(* Trigger ********************************************************)

(* Bausteine ******************************************************)
	Event													:	EventHandlingGrp10 := (
																	AutoConfirm			:= FALSE, 
																	SetClass 			:= TC2_SYSTEM.TCEVENTCLASS_ALARM );
	ChnEvent												:	NciChnEventHandling;

(* Dummy Speicher *************************************************)
	i														:	INT ;

END_VAR

(* Error message NCI channel to EventLogger 	V1.0	DS	*)
(***********************************************************)

(* Sequence **************************************************************)
IF __ISVALIDREF(rNci) 
THEN
	(* get Quit signal **************************************************)
	IF ConfirmTrig 
	THEN 
		QuitInternal 										:= TRUE; 
	END_IF (* set false see below *)

(* Event Logger Meldungen *****************************************************)
	Event.no[1].Flag 										:= rNci.IsEStopRequested;
	Event.no[2].Flag 										:= rNci.IsFeedFromBackupList;   
	Event.no[3].Flag 										:= rNci.IsMovingBackward;   
	
(*
	Event.no[4].Flag 										:= FALSE;
	Event.no[5].Flag 										:= FALSE;
	Event.no[6].Flag 										:= FALSE;
	Event.no[7].Flag 										:= FALSE;
	Event.no[8].Flag 										:= FALSE;
	Event.no[9].Flag 										:= FALSE;
	Event.no[10].Flag 										:= FALSE;
*)
(* workl Event Ctrl *************************************************)
	IF Event.no[1].Text2 <> Name OR Event.no[1].Text2 <> ''
	THEN
		//Init EventClass
		Event.no[1].eClass 									:= TC2_SYSTEM.TCEVENTCLASS_HINT;
		Event.no[2].eClass 									:= TC2_SYSTEM.TCEVENTCLASS_STATEINFO;
		Event.no[3].eClass 									:= TC2_SYSTEM.TCEVENTCLASS_STATEINFO;

		(* Init Name *)
		FOR i := Event.MIN_EVENT TO Event.MAX_EVENT DO
			Event.no[i].Text2								:= SEL(LEN(name)>1,CONCAT('Channel id:',DWORD_TO_STRING(rNci.NciToPlc.ChnId)),name);
		END_FOR
	END_IF

	Event(
		ConfirmTrig := ConfirmTrig,
		Disable		:= NOT Enable,
		SourceId	:= SourceId + rNci.NciToPlc.ChnId,
		Status	 	=> );	

(* Send ErrorId Message Text **********************************)
	ChnEvent(
		ConfirmTrig	:= NOT Enable OR QuitInternal OR ErrorId = 0 AND ChnEvent.State <> 0,
		Name		:= name,
		ChannelId	:= rNci.NciToPlc.ChnId,
		SourceId	:= Event.SourceId,
		Flag		:= ErrorId > 0 AND Enable,
		ErrorID		:= ErrorId,
		State		=> );

(* EventStatus *************************************************)
	Status													:= ChnEvent.Status OR Event.Status;
	NoOfActiveEvents										:= Event.NoOfActiveEvents + SEL(ChnEvent.Status.31 , 0, 1);

(* Error unkonw pointer or channel id *****************************)
ELSE
	NoOfActiveEvents										:= 0;
	ChnEvent(Flag := FALSE, ConfirmTrig := ChnEvent.State <> 0);
	Event(Disable := TRUE, Status =>  ); 
	Status													:= ChnEvent.Status OR Event.Status;
END_IF

(* Default reset Quit Internal *******************************)
	QuitInternal 											:= FALSE;

(**************************************************************)

METHOD PUBLIC confirm : bool  //Return value = TRUE if execution finished 
VAR_INPUT
END_VAR
QuitInternal 												:= TRUE;
confirm														:= TRUE;
END_METHOD

END_FUNCTION_BLOCK

// POUs/Motion/TF5100-NCI/02_Options/MFunctions/NciMFnc
{attribute 'no_check'}
FUNCTION_BLOCK NciMFnc
VAR_OUTPUT CONSTANT 
	MIN_M_FUNC												:	 UINT := 0;
	MAX_M_FUNC												:	 UINT := 159;
	
//Predefined M Functions
	M2_PRG_END												:	UINT := 2;
	M17_END_SUBROUTINE										:	UINT := 17;
	M30_PRG_END_WITH_ALL_MFUNC								:	UINT := 30; 
END_VAR                 									
VAR_INPUT               									
	ConfirmHsk												:	BOOL := FALSE; (* oder Methode benutzen *)
	FastMFuncReset											:	BOOL := FALSE; (* Signal Start Reser der unter FastMFuncNo angegebenen MFunc Nr. *)
	FastMFuncNo												:	UINT (MIN_M_FUNC..MAX_M_FUNC) := MIN_M_FUNC; (* Nr. der MFunktion die Resetet werden soll *)
	rNCIRef													:	REFERENCE TO NCI_REF := 0;
END_VAR                 									
VAR_OUTPUT              	
	HskReq													:	BOOL;
	HskId													:	UINT; 	
	CntActive												:	INT; //Count number of active M fucntions
	Active													:	BOOL; //Rising trigger M-Function active
	No														:	ARRAY[MIN_M_FUNC..MAX_M_FUNC] OF BOOL; (* Array of M-Functions *)
	rtNo													:	ARRAY[MIN_M_FUNC..MAX_M_FUNC] OF BOOL; (* rising trigger of M-Functions *)
END_VAR                     								
VAR
(* Zwischenspeicher ************************************************************)
	MemFnc													:	INT := -1;

(* Deklaration Trigger **********************************************************)

(* Zeiten ******************************************************************)

(* Bausteine ***************************************************************)
	ItpResetFastMFuncEx										:  ItpResetFastMFuncEx := (tTimeOut	:= DEFAULT_ADS_TIMEOUT);

(* Dummy Speicher **********************************************************)
	i														:	UINT := 0;
	OK														:	BOOL;
END_VAR

	(************************************************************************************)
	(*																					*)
	(*		B E C K H O F F   N E W   A U T O M A T I O N   T E C H N O L O G Y    		*)
	(*																					*)
	(*		Eiserstr.5	D-33415 Verl	Germany	phone:	+49-5246-0	www.Beckhoff.Com	*)
    (*																					*)
    (*		Bausteinbeschreibung	:	Auswerten von M-Funktionen						*)
	(*		TwinCAT-Version			:	2.11.x 											*)
	(*		Version					:	V2.0/ 05/20										*)
 	(*		Autor					:	Daniel Schlingmann								*)
	(*		Lib						:	TcNCI.Lib										*)
	(*																					*)
	(************************************************************************************)

(* evaluate M-function with additional acknowledge *********************************************************************)
	HskReq 													:= rNCIRef.NciToPlc.HskMFuncReq.0;
	HskId 													:= SEL(HskReq, 0, rNCIRef.NciToPlc.HskMFuncNo);

	(* Confirm request *)
	rNCIRef.PlcToNci.MFuncGranted.0 						:= (ConfirmHsk OR rNCIRef.PlcToNci.MFuncGranted.0) AND rNCIRef.NciToPlc.HskMFuncReq.0;

(* set all M-function setzen *)
	CntActive												:= 0;
	Active													:= FALSE;
	
	FOR i := MIN_M_FUNC TO MAX_M_FUNC DO
	 	OK	 												:= ItpIsFastMFunc(UINT_TO_INT(i),rNCIRef.NciToPlc) OR rNCIRef.NciToPlc.HskMFuncNo = i AND rNCIRef.NciToPlc.HskMFuncReq.0;
		rtNo[i]												:= NOT No[i] AND OK;
		No[i]												:= OK;
		IF No[i] 
		THEN 
			CntActive										:= CntActive + 1;		
			Active 											:= TRUE; 
		END_IF
	END_FOR

(* reset fast M-functions, ResetFastMFunc can also be used *)
	IF MemFnc < 0
	THEN
		IF FastMFuncReset
		THEN
			MemFnc 											:= 1;
			ResetFastMFunc(FastMFuncNo:= FastMFuncNo);
		END_IF
	ELSE 
		ResetFastMFunc(FastMFuncNo:= FastMFuncNo);		
	END_IF

(************************************************************************************)

METHOD PUBLIC confirm : BOOL //Return value = TRUE if execution finished
//required parameter
//rNCIRef
VAR_INPUT
END_VAR
IF __ISVALIDREF(rNCIRef)
THEN
	rNCIRef.PlcToNci.MFuncGranted.0 						:= rNCIRef.NciToPlc.HskMFuncReq.0;
	Confirm													:= NOT rNCIRef.NciToPlc.HskMFuncReq.0;
ELSE
	Confirm 												:= TRUE;
END_IF
END_METHOD

METHOD PUBLIC resetFastMFunc : BOOL //Return value = TRUE if busy
//required parameter
//rNCIRef
VAR_INPUT
	FastMFuncNo												:	UINT; (* number of M-function, which has to be resetted *)
END_VAR
IF NOT __ISVALIDREF(rNCIRef)
THEN
	ResetFastMFunc											:= FALSE;
	Return;	
END_IF

	IF ItpIsFastMFunc(UINT_TO_INT(FastMFuncNo),rNCIRef.NciToPlc) 
	THEN
		ItpResetFastMFuncEx.bExecute 						:= TRUE;
		MemFnc.0											:= TRUE;
	ELSIF NOT ItpResetFastMFuncEx.bBusy             		
	THEN                                            		
		ItpResetFastMFuncEx.bExecute 						:= FALSE;
	END_IF
	
	THIS^.FastMFuncNo										:= FastMFuncNo;

	ItpResetFastMFuncEx(
		bExecute	:= ,
		nMFuncNo	:= FastMFuncNo,
		tTimeOut	:= ,
		sNciToPlc	:= rNCIRef.NciToPlc,
		bBusy		=> ,
		bErr		=> ,
		nErrId	=> );
		
	IF NOT ItpResetFastMFuncEx.bBusy
	THEN
		IF ItpResetFastMFuncEx.bExecute
		THEN
			;
		//	Error											:=	ItpResetFastMFuncEx.bErr;
		//	ErrorId											:= ItpResetFastMFuncEx.nErrId;
		END_IF
		IF NOT ItpIsFastMFunc(UINT_TO_INT(FastMFuncNo),rNCIRef.NciToPlc) 
		THEN
			MemFnc											:= -1;
			ItpResetFastMFuncEx(bExecute := FALSE , sNciToPlc:= rNCIRef.NciToPlc);
		END_IF
	END_IF
	
	resetFastMFunc											:= ItpResetFastMFuncEx.bBusy;
END_METHOD

END_FUNCTION_BLOCK

// POUs/Motion/TF5100-NCI/02_Options/PlcItp/NciCreateItpTable
{attribute 'no_check'}
//Create Nci PlcInterpolation tabel
//
FUNCTION_BLOCK NciCreateItpTable
VAR_INPUT
	BlockNo													: UDINT := 0; //Block number addtional parameter for methods. At 0 -> block number will be automatically increased by every new entry
	OffsetFactorTblNumber									: UDINT := 100; 
	MaxTblNumber											: UDINT := 1000; 
END_VAR                     								
VAR_OUTPUT                  								
	Table													: ST_NciFeedGroupTable;
	FilledRows												: INT;
	LastBlockNo												: UDINT; //Last Blocknumber 
	Error													: BOOL;
{attribute 'displaymode':='hex'}
	ErrorID													: UDINT;
	ErrorText												: STRING(20);
END_VAR                     								
VAR
// Cache *******************************************
	TableNumber												: UDINT := 0;
	BlockCount												: UDINT := 1;

// Timer ******************************************************
// Trigger ****************************************************
// Blocks *****************************************************
	TblTemplate												: NciCreateItpTableEntryTemplate;
// Error ******************************************************
// Dummy Speicher *********************************************
	i														: INT := 0;
END_VAR

(* writing TcPlcInterpolation table				V1.5	*)
(********************************************************)

(* pleas use methods instead of the function-block body ********************)
	;
(***************************************************************************)

METHOD addCircleCIP : BOOL //Return value = TRUE if executed succesful
VAR_INPUT
	X														: LREAL := 0.0;
	Y														: LREAL := 0.0;
	Z														: LREAL := 0.0;
	Q1														: LREAL := 0.0;
	Q2														: LREAL := 0.0;
	Q3														: LREAL := 0.0;
	Q4														: LREAL := 0.0;
	Q5														: LREAL := 0.0;
	Velo													: LREAL; 	// mm/s 
	AccurateStop											: BOOL := FALSE;
	CIPPosX													: LREAL := 0.0;
	CIPPosY													: LREAL := 0.0;
	CIPPosZ													: LREAL := 0.0;
END_VAR
	(* NCI GeoCirclePlane schreiben									*)
	(*********************************************************)

(* Zielpos. in Tabelle schreiben ************************************************************)
	BlockCount 												:= BlockCount + 1;
	TblTemplate.GeoCircleCIP.nDisplayIndex := LastBlockNo 	:= SEL(BlockNo = 0, BlockNo, TableNumber * OffsetFactorTblNumber + BlockCount);
	TblTemplate.GeoCircleCIP.fEndPosX						:= X;
	TblTemplate.GeoCircleCIP.fEndPosY						:= Y;
	TblTemplate.GeoCircleCIP.fEndPosZ						:= Z;
	TblTemplate.GeoCircleCIP.fEndPosQ1						:= Q1;
	TblTemplate.GeoCircleCIP.fEndPosQ2						:= Q2;
	TblTemplate.GeoCircleCIP.fEndPosQ3						:= Q3;
	TblTemplate.GeoCircleCIP.fEndPosQ4						:= Q4;
	TblTemplate.GeoCircleCIP.fEndPosQ5						:= Q5;
	TblTemplate.GeoCircleCIP.fVelo							:= Velo;
	TblTemplate.GeoCircleCIP.bAccurateStop					:= AccurateStop;
	TblTemplate.GeoCircleCIP.fCIPPosX						:= CIPPosX;
	TblTemplate.GeoCircleCIP.fCIPPosY						:= CIPPosY;
	TblTemplate.GeoCircleCIP.fCIPPosZ						:= CIPPosZ;
                                                        	
	TblTemplate.InsertGeoCircleCIP(Table:= Table);    	
	Error													:= TblTemplate.Error;
	ErrorId													:= TblTemplate.ErrorId;
	ErrorText												:= TblTemplate.ErrorText;
	FilledRows												:= TblTemplate.FilledRows;

	AddCircleCip											:= NOT Error;
(***************************************************************************)
END_METHOD

METHOD addDwellTime : BOOL //Return value = TRUE if executed succesful
VAR_INPUT
	/// UCS ObjectID 
	Value													: LREAL ;
END_VAR
(*  													*)
(********************************************************)
	BlockCount 												:= BlockCount + 1;
	TblTemplate.DwellTime.nDisplayIndex	 := LastBlockNo 	:= SEL(BlockNo = 0, BlockNo, TableNumber * OffsetFactorTblNumber + BlockCount);
	TblTemplate.DwellTime.fDwellTime						:= Value;

	TblTemplate.InsertDwellTime(Table:= Table);
	Error													:= TblTemplate.Error;
	ErrorId													:= TblTemplate.ErrorId;
	ErrorText												:= TblTemplate.ErrorText;
	FilledRows												:= TblTemplate.FilledRows;

	AddDwellTime											:= not Error;	
	

(***************************************************************************)
END_METHOD

METHOD addEndOfTable : BOOL //Return value = TRUE if executed succesful
TblTemplate.InsertEndOfTable(Table:= Table);
Error													:= TblTemplate.Error;
ErrorId													:= TblTemplate.ErrorId;
ErrorText												:= TblTemplate.ErrorText;
FilledRows												:= TblTemplate.FilledRows;

AddEndOfTable											:= NOT Error;
END_METHOD

METHOD addMFuncFast : BOOL //Return value = TRUE if executed succesful
VAR_INPUT
	MFuncNo													: INT := 0;
END_VAR
(*														*)
(********************************************************)

(*************************************************************************************)
	BlockCount 												:= BlockCount + 1;
	TblTemplate.MFuncFast.nDisplayIndex := LastBlockNo 		:= SEL(BlockNo = 0, BlockNo, TableNumber * OffsetFactorTblNumber + BlockCount);
	TblTemplate.MFuncFast.nMFuncIn0							:= MFuncNo;
	TblTemplate.MFuncFast.nMFuncIn1							:= -1;
	TblTemplate.MFuncFast.nMFuncIn2							:= -1;
	TblTemplate.MFuncFast.nMFuncIn3							:= -1;
	TblTemplate.MFuncFast.nMFuncIn4							:= -1;
	TblTemplate.MFuncFast.nMFuncIn5							:= -1;
	TblTemplate.MFuncFast.nMFuncIn6							:= -1;
	TblTemplate.MFuncFast.nMFuncIn7							:= -1;
	
	TblTemplate.InsertMFuncFast(Table:= Table);
	Error													:= TblTemplate.Error;
	ErrorId													:= TblTemplate.ErrorId;
	ErrorText												:= TblTemplate.ErrorText;
	FilledRows												:= TblTemplate.FilledRows;
	
	AddMFuncFast											:= not Error;
(*************************************************************************************)
END_METHOD

METHOD addMFuncFastList : BOOL //Return value = TRUE if executed succesful
VAR_INPUT
	MFuncNo0												: INT := -1; //0-159 > Set to -1 to mark end of used MFunc
	MFuncNo1												: INT := -1; //0-159 > Set to -1 to mark end of used MFunc
	MFuncNo2												: INT := -1; //0-159 > Set to -1 to mark end of used MFunc
	MFuncNo3												: INT := -1; //0-159 > Set to -1 to mark end of used MFunc
	MFuncNo4												: INT := -1; //0-159 > Set to -1 to mark end of used MFunc
	MFuncNo5												: INT := -1; //0-159 > Set to -1 to mark end of used MFunc
	MFuncNo6												: INT := -1; //0-159 > Set to -1 to mark end of used MFunc
	MFuncNo7												: INT := -1; //0-159 > Set to -1 to mark end of used MFunc
END_VAR
(*														*)
(********************************************************)

(*************************************************************************************)
	BlockCount 												:= BlockCount + 1;
	TblTemplate.MFuncFast.nDisplayIndex := LastBlockNo 		:= SEL(BlockNo = 0, BlockNo, TableNumber * OffsetFactorTblNumber + BlockCount);
	TblTemplate.MFuncFast.nMFuncIn0							:= MFuncNo0;
	TblTemplate.MFuncFast.nMFuncIn1							:= MFuncNo1;
	TblTemplate.MFuncFast.nMFuncIn2							:= MFuncNo2;
	TblTemplate.MFuncFast.nMFuncIn3							:= MFuncNo3;
	TblTemplate.MFuncFast.nMFuncIn4							:= MFuncNo4;
	TblTemplate.MFuncFast.nMFuncIn5							:= MFuncNo5;
	TblTemplate.MFuncFast.nMFuncIn6							:= MFuncNo6;
	TblTemplate.MFuncFast.nMFuncIn7							:= MFuncNo7;
	
	TblTemplate.InsertMFuncFast(Table:= Table);
	Error													:= TblTemplate.Error;
	ErrorId													:= TblTemplate.ErrorId;
	ErrorText												:= TblTemplate.ErrorText;
	FilledRows												:= TblTemplate.FilledRows;
	
	AddMFuncFastList										:= NOT Error;
(*************************************************************************************)
END_METHOD

METHOD addMFuncHsk : BOOL //Return value = TRUE if executed succesful
VAR_INPUT
	MFuncNo													: INT := 0;
END_VAR
(* 														*)
(********************************************************)

(*************************************************************************************)
	BlockCount 												:= BlockCount + 1;
	TblTemplate.MFuncHsk.nDisplayIndex := LastBlockNo 		:= SEL(BlockNo = 0, BlockNo,  TableNumber * OffsetFactorTblNumber + BlockCount);
	TblTemplate.MFuncHsk.nMFunc								:= MFuncNo;
                                                        	
	TblTemplate.InsertMFuncHsk(Table:= Table);          	
	Error													:= TblTemplate.Error;
	ErrorId													:= TblTemplate.ErrorId;
	ErrorText												:= TblTemplate.ErrorText;
	FilledRows												:= TblTemplate.FilledRows;
	
	AddMFuncHsk												:= not Error;
(*************************************************************************************)
END_METHOD

METHOD addMFuncResetAllFast : BOOL //Return value = TRUE if executed succesful
VAR_INPUT
END_VAR
(* NCI ResetAllFastMFunc schreiben								*)
(*************************************************************************************)

(* confirmError all fast M-functions****************************************************)
	BlockCount 													:= BlockCount + 1;
	TblTemplate.MFuncResetAllFast.nDisplayIndex	:= LastBlockNo 	:= SEL(BlockNo = 0, BlockNo, TableNumber * OffsetFactorTblNumber + BlockCount);
	TblTemplate.InsertMFuncResetAllFast(Table:= Table);
	Error														:= TblTemplate.Error;
	ErrorId														:= TblTemplate.ErrorId;
	ErrorText													:= TblTemplate.ErrorText;
	FilledRows													:= TblTemplate.FilledRows;
	
	AddMFuncResetAllFast										:= not Error;
(*************************************************************************************)
END_METHOD

METHOD reset : BOOL //Return value = TRUE if execution finished
VAR_INPUT
END_VAR
TblTemplate.Reset(Table := Table);
FilledRows													:= 0;
BlockCount 													:= 0;
LastBlockNo													:= 0;
TableNumber 												:= TableNumber + 1;

IF TableNumber > MaxTblNumber 
THEN 
	TableNumber 											:= 1; 
END_IF

Error 														:= FALSE;
Errorid														:= 0;
ErrorText													:= '';
Reset														:= TRUE;
END_METHOD

METHOD setAxisDynamics : bool //Return value = TRUE if executed succesful
VAR_INPUT
	AxisNo													:	UDINT;
	Acc,Dec,Jerk											:	LREAL;
END_VAR
	(* NCI SetAxisDynamics schreiben						*)
	(*********************************************************)

(* Zielpos. in Tabelle schreiben ************************************************************)
	BlockCount 												:= BlockCount + 1;
	TblTemplate.AxisDynamics.nDisplayIndex := LastBlockNo := SEL(BlockNo = 0, BlockNo, TableNumber * OffsetFactorTblNumber + BlockCount);

	TblTemplate.AxisDynamics.nAxis 							:= AxisNo;
	TblTemplate.AxisDynamics.fDec							:= Dec;
	TblTemplate.AxisDynamics.fJerk							:= Jerk;
	TblTemplate.AxisDynamics.fAcc							:= Acc;
                                                        	
	TblTemplate.InsertAxisDynamics(Table:= Table);    	
	Error													:= TblTemplate.Error;
	ErrorId													:= TblTemplate.ErrorId;
	ErrorText												:= TblTemplate.ErrorText;
	FilledRows												:= TblTemplate.FilledRows;

	SetAxisDynamics											:= NOT Error;
(***************************************************************************)
END_METHOD

METHOD setBaseFrame : bool //Return value = TRUE if executed succesful
VAR_INPUT
    ShiftX													: LREAL;
    ShiftY													: LREAL;
    ShiftZ													: LREAL;
    RotX													: LREAL;
    RotY													: LREAL;
    RotZ													: LREAL;
    ShiftQ1													: LREAL;
    ShiftQ2													: LREAL;
    ShiftQ3													: LREAL;
    ShiftQ4													: LREAL;
    ShiftQ5													: LREAL;
END_VAR
	(* NCI SetBaseFrame schreiben						*)
	(*********************************************************)

(* Zielpos. in Tabelle schreiben ************************************************************)
	BlockCount 												:= BlockCount + 1;
	TblTemplate.BaseFrame.nDisplayIndex := LastBlockNo := SEL(BlockNo = 0, BlockNo, TableNumber * OffsetFactorTblNumber + BlockCount);

    TblTemplate.BaseFrame.fShiftX 							:= ShiftX;
    TblTemplate.BaseFrame.fShiftY							:= ShiftY;
    TblTemplate.BaseFrame.fShiftZ							:= ShiftZ;
    TblTemplate.BaseFrame.fRotX								:= RotX;
    TblTemplate.BaseFrame.fRotY								:= RotY;
    TblTemplate.BaseFrame.fRotZ								:= RotZ;
    TblTemplate.BaseFrame.fShiftQ1							:= ShiftQ1;
    TblTemplate.BaseFrame.fShiftQ2							:= ShiftQ2;
    TblTemplate.BaseFrame.fShiftQ3							:= ShiftQ3;
    TblTemplate.BaseFrame.fShiftQ4							:= ShiftQ4;
    TblTemplate.BaseFrame.fShiftQ5							:= ShiftQ5;
                       	
	TblTemplate.InsertBaseFrame(Table:= Table);    	
	Error													:= TblTemplate.Error;
	ErrorId													:= TblTemplate.ErrorId;
	ErrorText												:= TblTemplate.ErrorText;
	FilledRows												:= TblTemplate.FilledRows;

	SetBaseFrame											:= NOT Error;
(***************************************************************************)
END_METHOD

METHOD setCirclePlane : BOOL //Return value = TRUE if executed succesful
VAR_INPUT
	X														: LREAL := 0.0;
	Y														: LREAL := 0.0;
	Z														: LREAL := 0.0;
	Q1														: LREAL := 0.0;
	Q2														: LREAL := 0.0;
	Q3														: LREAL := 0.0;
	Q4														: LREAL := 0.0;
	Q5														: LREAL := 0.0;
	Velo													: LREAL; 	// mm/s 
	AccurateStop											: BOOL := FALSE;
	Clockwise												: BOOL := TRUE;
	Plane													: E_NciGeoPlane := E_NciGeoPlaneXY;
	CenterX													: LREAL := 0.0;
	CenterY													: LREAL := 0.0;
	CenterZ													: LREAL := 0.0;
END_VAR
	(* NCI GeoCirclePlane schreiben									*)
	(*********************************************************)

(* Zielpos. in Tabelle schreiben ************************************************************)
	BlockCount 												:= BlockCount + 1;
	TblTemplate.GeoCirclePlane.nDisplayIndex := LastBlockNo := SEL(BlockNo = 0, BlockNo, TableNumber * OffsetFactorTblNumber + BlockCount);
	TblTemplate.GeoCirclePlane.fEndPosX						:= X;
	TblTemplate.GeoCirclePlane.fEndPosY						:= Y;
	TblTemplate.GeoCirclePlane.fEndPosZ						:= Z;
	TblTemplate.GeoCirclePlane.fEndPosQ1					:= Q1;
	TblTemplate.GeoCirclePlane.fEndPosQ2					:= Q2;
	TblTemplate.GeoCirclePlane.fEndPosQ3					:= Q3;
	TblTemplate.GeoCirclePlane.fEndPosQ4					:= Q4;
	TblTemplate.GeoCirclePlane.fEndPosQ5					:= Q5;
	TblTemplate.GeoCirclePlane.fVelo						:= Velo;
	TblTemplate.GeoCirclePlane.bAccurateStop				:= AccurateStop;
	TblTemplate.GeoCirclePlane.bClockwise					:= Clockwise;
	TblTemplate.GeoCirclePlane.nPlane						:= Plane;
	TblTemplate.GeoCirclePlane.fCenterX						:= CenterX;
	TblTemplate.GeoCirclePlane.fCenterY						:= CenterY;
	TblTemplate.GeoCirclePlane.fCenterZ						:= CenterZ;
                                                        	
	TblTemplate.InsertGeoCirclePlane(Table:= Table);    	
	Error													:= TblTemplate.Error;
	ErrorId													:= TblTemplate.ErrorId;
	ErrorText												:= TblTemplate.ErrorText;
	FilledRows												:= TblTemplate.FilledRows;

	SetCirclePlane											:= NOT Error;
(***************************************************************************)
END_METHOD

METHOD setCoordinateSystem : BOOL //Return value = TRUE if executed succesful
VAR_INPUT
	/// UCS ObjectID 
	ObjectId												: UDINT := 0;
END_VAR
(* NCI UserKos schreiben															*)
(************************************************************************************)

(* User Koordinatensystem schreiben ************************************************************)
	BlockCount 												:= BlockCount + 1;
	TblTemplate.SetCoordinateSystem.nDisplayIndex := LastBlockNo := SEL(BlockNo = 0, BlockNo, TableNumber * OffsetFactorTblNumber + BlockCount);
	TblTemplate.SetCoordinateSystem.nObjectId				:= ObjectId;

	TblTemplate.InsertSetCoordinateSystem(Table:= Table);
	Error													:= TblTemplate.Error;
	ErrorId													:= TblTemplate.ErrorId;
	ErrorText												:= TblTemplate.ErrorText;
	FilledRows												:= TblTemplate.FilledRows;
	
	SetCoordinateSystem										:= not Error;
(*************************************************************************************)
END_METHOD

METHOD setDynOverride : BOOL //Return value = TRUE if executed succesful
VAR_INPUT
	/// UCS ObjectID 
	Value													: lreal := 0; //0.0-100.0%
END_VAR
(* NCI Oevrride schreiben											*)
(********************************************************************)

(* insert override **************************************************)
	(* apapt override *)
	BlockCount 												:= BlockCount + 1;
	TblTemplate.DynOverride.nDisplayIndex := LastBlockNo 		:= SEL(BlockNo = 0, BlockNo, TableNumber * OffsetFactorTblNumber + BlockCount);
	TblTemplate.DynOverride.fDynOvr								:= 0.01 * Value;

	TblTemplate.InsertDynOverride(Table:= Table);
	Error													:= TblTemplate.Error;
	ErrorId													:= TblTemplate.ErrorId;
	ErrorText												:= TblTemplate.ErrorText;
	FilledRows												:= TblTemplate.FilledRows;
	
	SetDynOverride											:= not Error;
(*************************************************************************************)
END_METHOD

METHOD setGeoBezier3 : booL //Return value = TRUE if executed succesful
VAR_INPUT
     ControlPoint1X											: LREAL;
     ControlPoint1Y											: LREAL;
     ControlPoint1Z											: LREAL;
     ControlPoint2X											: LREAL;
     ControlPoint2Y											: LREAL;
     ControlPoint2Z											: LREAL;
     EndPosX												: LREAL;
     EndPosY												: LREAL;
     EndPosZ												: LREAL;
     EndPosQ1												: LREAL;
     EndPosQ2												: LREAL;
     EndPosQ3												: LREAL;
     EndPosQ4												: LREAL;
     EndPosQ5												: LREAL;
     Velo													: LREAL;
     AccurateStop											: BOOL; (* VeloEnd := 0 *)
END_VAR
	(* NCI SetGeoBezier3 schreiben						*)
	(*********************************************************)

(* Zielpos. in Tabelle schreiben ************************************************************)
	BlockCount 												:= BlockCount + 1;
	TblTemplate.GeoBezier3.nDisplayIndex := LastBlockNo := SEL(BlockNo = 0, BlockNo, TableNumber * OffsetFactorTblNumber + BlockCount);

    TblTemplate.GeoBezier3.fControlPoint1X					:= ControlPoint1X;
    TblTemplate.GeoBezier3.fControlPoint1Y					:= ControlPoint1Y;
    TblTemplate.GeoBezier3.fControlPoint1Z					:= ControlPoint1Z;
    TblTemplate.GeoBezier3.fControlPoint2X					:= ControlPoint2X;
    TblTemplate.GeoBezier3.fControlPoint2Y					:= ControlPoint2Y;
    TblTemplate.GeoBezier3.fControlPoint2Z					:= ControlPoint2Z;
    TblTemplate.GeoBezier3.fEndPosX							:= EndPosX;
    TblTemplate.GeoBezier3.fEndPosY							:= EndPosY;
    TblTemplate.GeoBezier3.fEndPosZ							:= EndPosZ;
    TblTemplate.GeoBezier3.fEndPosQ1						:= EndPosQ1;
    TblTemplate.GeoBezier3.fEndPosQ2						:= EndPosQ2;
    TblTemplate.GeoBezier3.fEndPosQ3						:= EndPosQ3;
    TblTemplate.GeoBezier3.fEndPosQ4						:= EndPosQ4;
    TblTemplate.GeoBezier3.fEndPosQ5						:= EndPosQ5;
    TblTemplate.GeoBezier3.fVelo							:= Velo;
    TblTemplate.GeoBezier3.bAccurateStop					:= AccurateStop  ;                            	
	
	TblTemplate.InsertGeoBezier3(Table:= Table);    	
	Error													:= TblTemplate.Error;
	ErrorId													:= TblTemplate.ErrorId;
	ErrorText												:= TblTemplate.ErrorText;
	FilledRows												:= TblTemplate.FilledRows;

	SetGeoBezier3											:= NOT Error;
(***************************************************************************)
END_METHOD

METHOD setGeoBezier5 : booL //Return value = TRUE if executed succesful
VAR_INPUT
     ControlPoint1X											: LREAL;
     ControlPoint1Y											: LREAL;
     ControlPoint1Z											: LREAL;
     ControlPoint2X											: LREAL;
     ControlPoint2Y											: LREAL;
     ControlPoint2Z											: LREAL;
     ControlPoint3X											: LREAL;
     ControlPoint3Y											: LREAL;
     ControlPoint3Z											: LREAL;
     ControlPoint4X											: LREAL;
     ControlPoint4Y											: LREAL;
     ControlPoint4Z											: LREAL;
     EndPosX												: LREAL;
     EndPosY												: LREAL;
     EndPosZ												: LREAL;
     EndPosQ1												: LREAL;
     EndPosQ2												: LREAL;
     EndPosQ3												: LREAL;
     EndPosQ4												: LREAL;
     EndPosQ5												: LREAL;
     Velo													: LREAL;
     AccurateStop											: BOOL; (* VeloEnd := 0 *)
END_VAR
	(* NCI SetGeoBezier5 schreiben						*)
	(*********************************************************)

(* Zielpos. in Tabelle schreiben ************************************************************)
	BlockCount 												:= BlockCount + 1;
	TblTemplate.GeoBezier5.nDisplayIndex := LastBlockNo := SEL(BlockNo = 0, BlockNo, TableNumber * OffsetFactorTblNumber + BlockCount);

    TblTemplate.GeoBezier5.fControlPoint1X					:= ControlPoint1X;
    TblTemplate.GeoBezier5.fControlPoint1Y					:= ControlPoint1Y;
    TblTemplate.GeoBezier5.fControlPoint1Z					:= ControlPoint1Z;
    TblTemplate.GeoBezier5.fControlPoint2X					:= ControlPoint2X;
    TblTemplate.GeoBezier5.fControlPoint2Y					:= ControlPoint2Y;
    TblTemplate.GeoBezier5.fControlPoint2Z					:= ControlPoint2Z;
    TblTemplate.GeoBezier5.fControlPoint3X					:= ControlPoint3X;
    TblTemplate.GeoBezier5.fControlPoint3Y					:= ControlPoint3Y;
    TblTemplate.GeoBezier5.fControlPoint3Z					:= ControlPoint3Z;
    TblTemplate.GeoBezier5.fControlPoint4X					:= ControlPoint4X;
    TblTemplate.GeoBezier5.fControlPoint4Y					:= ControlPoint4Y;
    TblTemplate.GeoBezier5.fControlPoint4Z					:= ControlPoint4Z;
    TblTemplate.GeoBezier5.fEndPosX							:= EndPosX;
    TblTemplate.GeoBezier5.fEndPosY							:= EndPosY;
    TblTemplate.GeoBezier5.fEndPosZ							:= EndPosZ;
    TblTemplate.GeoBezier5.fEndPosQ1						:= EndPosQ1;
    TblTemplate.GeoBezier5.fEndPosQ2						:= EndPosQ2;
    TblTemplate.GeoBezier5.fEndPosQ3						:= EndPosQ3;
    TblTemplate.GeoBezier5.fEndPosQ4						:= EndPosQ4;
    TblTemplate.GeoBezier5.fEndPosQ5						:= EndPosQ5;
    TblTemplate.GeoBezier5.fVelo							:= Velo;
    TblTemplate.GeoBezier5.bAccurateStop					:= AccurateStop  ;                            	
	
	TblTemplate.InsertGeoBezier5(Table:= Table);    	
	Error													:= TblTemplate.Error;
	ErrorId													:= TblTemplate.ErrorId;
	ErrorText												:= TblTemplate.ErrorText;
	FilledRows												:= TblTemplate.FilledRows;

	SetGeoBezier5											:= NOT Error;
(***************************************************************************)
END_METHOD

METHOD setGeoLine : BOOL //Return value = TRUE if executed succesful
VAR_INPUT
	X														: LREAL := 0.0;
	Y														: LREAL := 0.0;
	Z														: LREAL := 0.0;
	Q1														: LREAL := 0.0;
	Q2														: LREAL := 0.0;
	Q3														: LREAL := 0.0;
	Q4														: LREAL := 0.0;
	Q5														: LREAL := 0.0;
	Velo													: LREAL; 	// mm/s 
	AccurateStop											: BOOL := FALSE;
END_VAR
(* writing NCI GeoLine 									*)
(********************************************************)

(***************************************************************************)
	BlockCount 												:= BlockCount + 1;
	TblTemplate.GeoLine.nDisplayIndex := LastBlockNo 		:= SEL(BlockNo = 0, BlockNo, TableNumber * OffsetFactorTblNumber + BlockCount);
	TblTemplate.GeoLine.fEndPosX							:= X;
	TblTemplate.GeoLine.fEndPosY							:= Y;
	TblTemplate.GeoLine.fEndPosZ							:= Z;
	TblTemplate.GeoLine.fEndPosQ1							:= Q1 ;
	TblTemplate.GeoLine.fEndPosQ2							:= Q2;
	TblTemplate.GeoLine.fEndPosQ3							:= Q3;
	TblTemplate.GeoLine.fEndPosQ4							:= Q4;
	TblTemplate.GeoLine.fEndPosQ5							:= Q5;
	TblTemplate.GeoLine.fVelo								:= Velo;
	TblTemplate.GeoLine.bRapidTraverse						:= Velo = 0.0;
	TblTemplate.GeoLine.bAccurateStop						:= AccurateStop;
                                                        	
	TblTemplate.InsertGeoLine(Table:= Table);           	
	Error													:= TblTemplate.Error;
	ErrorId													:= TblTemplate.ErrorId;
	ErrorText												:= TblTemplate.ErrorText;
	FilledRows												:= TblTemplate.FilledRows;
	
	SetGeoLine												:= not Error;
(***************************************************************************)
END_METHOD

METHOD setGeoStart : BOOL //Return value = TRUE if executed succesful
VAR_INPUT
	X														: LREAL := 0.0;
	Y														: LREAL := 0.0;
	Z														: LREAL := 0.0;
	Q1														: LREAL := 0.0;
	Q2														: LREAL := 0.0;
	Q3														: LREAL := 0.0;
	Q4														: LREAL := 0.0;
	Q5														: LREAL := 0.0;
END_VAR
(* writing NCI GeoLine 									*)
(********************************************************)

(***************************************************************************)
	TblTemplate.GeoStart.fPosX								:= X;
	TblTemplate.GeoStart.fPosY								:= Y;
	TblTemplate.GeoStart.fPosZ								:= Z;
	TblTemplate.GeoStart.fPosQ1								:= Q1 ;
	TblTemplate.GeoStart.fPosQ2								:= Q2;
	TblTemplate.GeoStart.fPosQ3								:= Q3;
	TblTemplate.GeoStart.fPosQ4								:= Q4;
	TblTemplate.GeoStart.fPosQ5								:= Q5;
                                                        	
	TblTemplate.InsertGeoStart(Table:= Table);           	
	Error													:= TblTemplate.Error;
	ErrorId													:= TblTemplate.ErrorId;
	ErrorText												:= TblTemplate.ErrorText;
	FilledRows												:= TblTemplate.FilledRows;
	
	SetGeoStart												:= not Error;
(***************************************************************************)
END_METHOD

METHOD setHParam : booL //Return value = TRUE if executed succesful
VAR_INPUT
	HParam													: UDINT;
END_VAR
(* 														*)
(********************************************************)

(*************************************************************************************)
	BlockCount 												:= BlockCount + 1;
	TblTemplate.HParam.nDisplayIndex := LastBlockNo 		:= SEL(BlockNo = 0, BlockNo,  TableNumber * OffsetFactorTblNumber + BlockCount);
	TblTemplate.HParam.nHParam								:= HParam;
                                                        	
	TblTemplate.InsertHParam(Table:= Table);          	
	Error													:= TblTemplate.Error;
	ErrorId													:= TblTemplate.ErrorId;
	ErrorText												:= TblTemplate.ErrorText;
	FilledRows												:= TblTemplate.FilledRows;
	
	SetHParam												:= NOT Error;
(*************************************************************************************)
END_METHOD

METHOD setPathDynamics : BOOL //Return value = TRUE if executed succesful
VAR_INPUT
	Acc,Dec,Jerk											:	LREAL;
END_VAR
	(* NCI SetPathDynamics schreiben						*)
	(*********************************************************)

(* Zielpos. in Tabelle schreiben ************************************************************)
	BlockCount 												:= BlockCount + 1;
	TblTemplate.PathDynamics.nDisplayIndex := LastBlockNo := SEL(BlockNo = 0, BlockNo, TableNumber * OffsetFactorTblNumber + BlockCount);

	TblTemplate.PathDynamics.fDec							:= Dec;
	TblTemplate.PathDynamics.fJerk							:= Jerk;
	TblTemplate.PathDynamics.fAcc							:= Acc;
                                                        	
	TblTemplate.InsertPathDynamics(Table:= Table);    	
	Error													:= TblTemplate.Error;
	ErrorId													:= TblTemplate.ErrorId;
	ErrorText												:= TblTemplate.ErrorText;
	FilledRows												:= TblTemplate.FilledRows;

	SetPathDynamics											:= NOT Error;
(***************************************************************************)
END_METHOD

METHOD setSParam : bool //Return value = TRUE if executed succesful
VAR_INPUT
	SParam													: UINT;
END_VAR
(* 														*)
(********************************************************)

(*************************************************************************************)
	BlockCount 												:= BlockCount + 1;
	TblTemplate.SParam.nDisplayIndex := LastBlockNo 		:= SEL(BlockNo = 0, BlockNo,  TableNumber * OffsetFactorTblNumber + BlockCount);
	TblTemplate.SParam.nSParam								:= SParam;
                                                        	
	TblTemplate.InsertSParam(Table:= Table);          	
	Error													:= TblTemplate.Error;
	ErrorId													:= TblTemplate.ErrorId;
	ErrorText												:= TblTemplate.ErrorText;
	FilledRows												:= TblTemplate.FilledRows;
	
	SetSParam												:= NOT Error;
(*************************************************************************************)
END_METHOD

METHOD setTangFollowingDesc : booL //Return value = TRUE if executed succesful
VAR_INPUT
    TangOn													: BOOL;
    TangAxis												: E_NciAxesInGroup;  
    PathAxis1												: E_NciAxesInGroup; 
    PathAxis2												: E_NciAxesInGroup; 
    Offset													: LREAL; 
    CriticalAngle1											: LREAL;
    TfBehavior												: E_TangentialFollowingBehavior; 
END_VAR
	(* NCI SetTangFollowingDesc schreiben						*)
	(*********************************************************)

(* Zielpos. in Tabelle schreiben ************************************************************)
	BlockCount 												:= BlockCount + 1;
	LastBlockNo 											:= SEL(BlockNo = 0, BlockNo, TableNumber * OffsetFactorTblNumber + BlockCount);

    TblTemplate.TangentialFollowingDesc.bTangOn				:= TangOn;
    TblTemplate.TangentialFollowingDesc.nTangAxis			:= TangAxis;
    TblTemplate.TangentialFollowingDesc.nPathAxis1			:= PathAxis1;
    TblTemplate.TangentialFollowingDesc.nPathAxis2			:= PathAxis2;
    TblTemplate.TangentialFollowingDesc.fOffset				:= Offset;
    TblTemplate.TangentialFollowingDesc.fCriticalAngle1		:= CriticalAngle1;
    TblTemplate.TangentialFollowingDesc.nTfBehavior			:= TfBehavior;
                       	
	TblTemplate.InsertTangFollowingDesc(Table:= Table);    	
	Error													:= TblTemplate.Error;
	ErrorId													:= TblTemplate.ErrorId;
	ErrorText												:= TblTemplate.ErrorText;
	FilledRows												:= TblTemplate.FilledRows;

	SetTangFollowingDesc									:= NOT Error;
(***************************************************************************)
END_METHOD

METHOD setTParam : bool //Return value = TRUE if executed succesful
VAR_INPUT
	TParam													: UINT;
END_VAR
(* 														*)
(********************************************************)

(*************************************************************************************)
	BlockCount 												:= BlockCount + 1;
	TblTemplate.TParam.nDisplayIndex := LastBlockNo 		:= SEL(BlockNo = 0, BlockNo,  TableNumber * OffsetFactorTblNumber + BlockCount);
	TblTemplate.TParam.nTParam								:= TParam;
                                                        	
	TblTemplate.InsertTParam(Table:= Table);          	
	Error													:= TblTemplate.Error;
	ErrorId													:= TblTemplate.ErrorId;
	ErrorText												:= TblTemplate.ErrorText;
	FilledRows												:= TblTemplate.FilledRows;
	
	SetTParam												:= NOT Error;
(**************************************************************************)
END_METHOD

METHOD setVertexSmoothing : BOOL //Return value = TRUE if executed succesful
VAR_INPUT
	Radius													: LREAL := 0.0;
	VertSmType												: UDINT := 5;
	VertSmSubType											: UDINT := 3;
END_VAR
(* writing NCI Vertex smoothing 								*)
(****************************************************************)

(* writing into table	*****************************************)
	BlockCount 												:= BlockCount + 1;
	TblTemplate.VertexSmoothing.nDisplayIndex := LastBlockNo := SEL(BlockNo = 0, BlockNo, TableNumber * OffsetFactorTblNumber + BlockCount);
	TblTemplate.VertexSmoothing.nType						:= VertSmType;
	TblTemplate.VertexSmoothing.nSubtype					:= VertSmSubtype; (* 	1: constant radius tolerance
																					2: distance between Abstand intersectoin point and peal point
																					3: adaptiv raidus tolerance
																					*)
	TblTemplate.VertexSmoothing.fRadius						:= Radius; (* mm *)

	TblTemplate.InsertVertexSmoothing(Table:= Table);
	Error													:= TblTemplate.Error;
	ErrorId													:= TblTemplate.ErrorId;
	ErrorText												:= TblTemplate.ErrorText;
	FilledRows												:= TblTemplate.FilledRows;
	SetVertexSmoothing										:= not Error;
(*************************************************************************************)
END_METHOD

END_FUNCTION_BLOCK

// POUs/Motion/TF5100-NCI/02_Options/PlcItp/NciCreateItpTableEntryTemplate
FUNCTION_BLOCK NciCreateItpTableEntryTemplate
VAR_INPUT
	EndOfTables												: ST_NciEndOfTables;
	GeoCirclePlane											: ST_NciGeoCirclePlane;
	GeoCircleCIP											: ST_NciGeoCircleCIP;
	GeoLine													: ST_NciGeoLine;
	GeoBezier3												: ST_NciGeoBezier3;
	GeoBezier5												: ST_NciGeoBezier5;	
	GeoStart												: ST_NciGeoStart;
	TangentialFollowingDesc									: ST_NciTangentialFollowingDesc;
	MFuncHsk												: ST_NciMFuncHsk;
	MFuncFast												: ST_NciMFuncFast;
	MFuncResetAllFast										: ST_NciMFuncResetAllFast;
	HParam													: ST_NciHParam;
	SParam													: ST_NciSParam;
	TParam													: ST_NciTParam;
	DynOverride												: ST_NciDynOvr;
	VertexSmoothing											: ST_NciVertexSmoothing;
	PathDynamics											: ST_NciPathDynamics;
	BaseFrame												: ST_NciBaseFrame;
	SetCoordinateSystem										: ST_NciSetCoordinateSystem;
	AxisDynamics											: ST_NciAxisDynamics;
	DwellTime												: ST_NciDwellTime;
END_VAR
VAR_OUTPUT
	FilledRows												: INT;
	Error													: BOOL;
{attribute 'displaymode':='hex'}
	ErrorId													: UDINT;
	ErrorText												: STRING(20);
END_VAR                 									
VAR                     									
	TblPrep													: FB_NciFeedTablePreparation;
END_VAR

(* NCI Table entry template				 	V2.0	*)
(****************************************************)

(******************************************************************************)
;
(******************************************************************************)

METHOD insertAxisDynamics : bool //Return value = TRUE if executed succesful
VAR_IN_OUT
	Table													: ST_NciFeedGroupTable;
END_VAR
	TblPrep(
		nEntryType			:= AxisDynamics.nEntryType,
		pEntry				:= ADR(AxisDynamics),
		stFeedGroupTable	:= Table,
		nFilledRows			=> FilledRows,
		bError				=> ,
		nErrorId			=> );

	IF TblPrep.bError 
	THEN
		Error												:= TRUE;
		ErrorText											:= CONCAT('AxisDynamics - JobNo. :',UDINT_TO_STRING(AxisDynamics.nDisplayIndex));
		ErrorId												:= TblPrep.nErrorId;
	ELSE
		insertAxisDynamics									:= TRUE;
	END_IF
END_METHOD

METHOD insertBaseFrame : bool //Return value = TRUE if executed succesful
VAR_IN_OUT
	Table													: ST_NciFeedGroupTable;
END_VAR
	TblPrep(
		nEntryType		:= BaseFrame.nEntryType,
		pEntry			:= ADR(BaseFrame),
		stFeedGroupTable:= Table,
		nFilledRows		=> FilledRows,
		bError			=> ,
		nErrorId		=> );

	IF TblPrep.bError 
	THEN
		Error												:= TRUE;
		ErrorText											:= CONCAT('BaseFrame - JobNo. :',UDINT_TO_STRING(BaseFrame.nDisplayIndex));
		ErrorId												:= TblPrep.nErrorId;
	ELSE
		insertBaseFrame										:= TRUE;
	END_IF
END_METHOD

METHOD insertDwellTime : booL //Return value = TRUE if executed succesful
VAR_IN_OUT
	Table													: ST_NciFeedGroupTable;
END_VAR
	TblPrep(
		nEntryType		:= DwellTime.nEntryType,
		pEntry			:= ADR(DwellTime),
		stFeedGroupTable:= Table,
		nFilledRows		=> FilledRows,
		bError			=> ,
		nErrorId		=> );

	IF TblPrep.bError 
	THEN
		Error												:= TRUE;
		ErrorText											:= CONCAT('DwellTime - JobNo. :',UDINT_TO_STRING(DwellTime.nDisplayIndex));
		ErrorId												:= TblPrep.nErrorId;
	ELSE
		insertDwellTime										:= TRUE;
	END_IF
END_METHOD

METHOD insertDynOverride : booL //Return value = TRUE if executed succesful
VAR_IN_OUT
	Table													: ST_NciFeedGroupTable;
END_VAR
	TblPrep(
		nEntryType			:= DynOverride.nEntryType,
		pEntry				:= ADR(DynOverride),
		stFeedGroupTable	:= Table,
		nFilledRows			=> FilledRows,
		bError				=> ,
		nErrorId			=> );

	IF TblPrep.bError THEN
		Error												:= TRUE;
		ErrorText											:= CONCAT('DynOverride - JobNo. :',UDINT_TO_STRING(DynOverride.nDisplayIndex));
		ErrorId												:= TblPrep.nErrorId;
	ELSE
		insertDynOverride									:= TRUE;
	END_IF
END_METHOD

METHOD insertEndOfTable : bool //Return value = TRUE if executed succesful
VAR_IN_OUT
	Table													: ST_NciFeedGroupTable;
END_VAR
	TblPrep(
		nEntryType			:= EndOfTables.nEntryType,
		pEntry				:= ADR(EndOfTables),
		stFeedGroupTable	:= Table,
		nFilledRows			=> FilledRows,
		bError				=> ,
		nErrorId			=> );

	IF TblPrep.bError THEN
		Error												:= TRUE;
		ErrorText											:= CONCAT('EndOfTables - FilledRows :',INT_TO_STRING(FilledRows));
		ErrorId												:= TblPrep.nErrorId;
	ELSE
		insertEndOfTable									:= TRUE;
	END_IF
END_METHOD

METHOD insertGeoBezier3 : booL //Return value = TRUE if executed succesful
VAR_IN_OUT
	Table													: ST_NciFeedGroupTable;
END_VAR
	TblPrep(
		nEntryType			:= GeoBezier3.nEntryType,
		pEntry				:= ADR(GeoBezier3),
		stFeedGroupTable	:= Table,
		nFilledRows			=> FilledRows,
		bError				=> ,
		nErrorId			=> );

	IF TblPrep.bError THEN
		Error												:= TRUE;
		ErrorText											:= CONCAT('GeoBezier3 - JobNo. :',UDINT_TO_STRING(GeoBezier3.nDisplayIndex));
		ErrorId												:= TblPrep.nErrorId;
	ELSE
		insertGeoBezier3									:= TRUE;
	END_IF
END_METHOD

METHOD insertGeoBezier5 : booL //Return value = TRUE if executed succesful
VAR_IN_OUT
	Table													: ST_NciFeedGroupTable;
END_VAR
	TblPrep(
		nEntryType			:= GeoBezier5.nEntryType,
		pEntry				:= ADR(GeoBezier5),
		stFeedGroupTable	:= Table,
		nFilledRows			=> FilledRows,
		bError				=> ,
		nErrorId			=> );

	IF TblPrep.bError THEN
		Error												:= TRUE;
		ErrorText											:= CONCAT('GeoBezier5 - JobNo. :',UDINT_TO_STRING(GeoBezier5.nDisplayIndex));
		ErrorId												:= TblPrep.nErrorId;
	ELSE
		insertGeoBezier5									:= TRUE;
	END_IF
END_METHOD

METHOD insertGeoCircleCIP : booL //Return value = TRUE if executed succesful
VAR_IN_OUT
	Table													: ST_NciFeedGroupTable;
END_VAR
	TblPrep(
		nEntryType			:= GeoCircleCIP.nEntryType,
		pEntry				:= ADR(GeoCircleCIP),
		stFeedGroupTable	:= Table,
		nFilledRows			=> FilledRows,
		bError				=> ,
		nErrorId			=> );

	IF TblPrep.bError 
	THEN
		Error												:= TRUE;
		ErrorText											:= CONCAT('GeoCircleCIP - JobNo. :',UDINT_TO_STRING(GeoCirclePlane.nDisplayIndex));
		ErrorId												:= TblPrep.nErrorId;
	ELSE
		insertGeoCircleCIP									:= TRUE;
	END_IF
END_METHOD

METHOD insertGeoCirclePlane : BOOL //Return value = TRUE if executed succesful
VAR_IN_OUT
	Table													: ST_NciFeedGroupTable;
END_VAR
	TblPrep(
		nEntryType			:= GeoCirclePlane.nEntryType,
		pEntry				:= ADR(GeoCirclePlane),
		stFeedGroupTable	:= Table,
		nFilledRows			=> FilledRows,
		bError				=> ,
		nErrorId			=> );

	IF TblPrep.bError 
	THEN
		Error												:= TRUE;
		ErrorText											:= CONCAT('GeoCirclePlane - JobNo. :',UDINT_TO_STRING(GeoCirclePlane.nDisplayIndex));
		ErrorId												:= TblPrep.nErrorId;
	ELSE
		insertGeoCirclePlane								:= TRUE;
	END_IF
END_METHOD

METHOD insertGeoLine : boOL //Return value = TRUE if executed succesful
VAR_IN_OUT
	Table													: ST_NciFeedGroupTable;
END_VAR
	TblPrep(
		nEntryType			:= GeoLine.nEntryType,
		pEntry				:= ADR(GeoLine),
		stFeedGroupTable	:= Table,
		nFilledRows			=> FilledRows,
		bError				=> ,
		nErrorId			=> );

	IF TblPrep.bError 
	THEN
		Error												:= TRUE;
		ErrorText											:= CONCAT('GeoLine - JobNo. :',UDINT_TO_STRING(GeoLine.nDisplayIndex));
		ErrorId												:= TblPrep.nErrorId;
	ELSE
		insertGeoLine										:= TRUE;
	END_IF
END_METHOD

METHOD insertGeoStart : booL //Return value = TRUE if executed succesful
VAR_IN_OUT
	Table													: ST_NciFeedGroupTable;
END_VAR
	TblPrep(
		nEntryType			:= GeoStart.nEntryType,
		pEntry				:= ADR(GeoStart),
		stFeedGroupTable	:= Table,
		nFilledRows			=> FilledRows,
		bError				=> ,
		nErrorId			=> );

	IF TblPrep.bError 
	THEN
		Error												:= TRUE;
		ErrorText											:= CONCAT('GeoStart - FilledRows. :',INT_TO_STRING(FilledRows));
		ErrorId												:= TblPrep.nErrorId;
	ELSE
		insertGeoStart										:= TRUE;
	END_IF
END_METHOD

METHOD insertHParam : booL //Return value = TRUE if executed succesful
VAR_IN_OUT
	Table													: ST_NciFeedGroupTable;
END_VAR
	TblPrep(
		nEntryType			:= HParam.nEntryType,
		pEntry				:= ADR(HParam),
		stFeedGroupTable	:= Table,
		nFilledRows			=> FilledRows,
		bError				=> ,
		nErrorId			=> );

	IF TblPrep.bError 
	THEN
		Error												:= TRUE;
		ErrorText											:= CONCAT('HParam - JobNo. :',UDINT_TO_STRING(HParam.nDisplayIndex));
		ErrorId												:= TblPrep.nErrorId;
	ELSE
		insertHParam										:= TRUE;
	END_IF
END_METHOD

METHOD insertMFuncFast : booL //Return value = TRUE if executed succesful
VAR_IN_OUT
	Table													: ST_NciFeedGroupTable;
END_VAR
	TblPrep(
		nEntryType			:= MFuncFast.nEntryType,
		pEntry				:= ADR(MFuncFast),
		stFeedGroupTable	:= Table,
		nFilledRows			=> FilledRows,
		bError				=> ,
		nErrorId			=> );

	IF TblPrep.bError 
	THEN
		Error												:= TRUE;
		ErrorText											:= CONCAT('MFuncFastList - JobNo. :',UDINT_TO_STRING(MFuncFast.nDisplayIndex));
		ErrorId												:= TblPrep.nErrorId;
	ELSE
		insertMFuncFast										:= TRUE;
	END_IF
END_METHOD

METHOD insertMFuncHsk : bool //Return value = TRUE if executed succesful
VAR_IN_OUT
	Table													: ST_NciFeedGroupTable;
END_VAR
	TblPrep(
		nEntryType			:= MFuncHsk.nEntryType,
		pEntry				:= ADR(MFuncHsk),
		stFeedGroupTable	:= Table,
		nFilledRows			=> FilledRows,
		bError				=> ,
		nErrorId			=> );

	IF TblPrep.bError 
	THEN
		Error												:= TRUE;
		ErrorText											:= CONCAT('MFuncHsk - JobNo. :',UDINT_TO_STRING(MFuncHsk.nDisplayIndex));
		ErrorId												:= TblPrep.nErrorId;
	ELSE
		insertMFuncHsk										:= TRUE;
	END_IF
END_METHOD

METHOD insertMFuncResetAllFast : bool //Return value = TRUE if executed succesful
VAR_IN_OUT
	Table													: ST_NciFeedGroupTable;
END_VAR
	TblPrep(
		nEntryType			:= MFuncResetAllFast.nEntryType,
		pEntry				:= ADR(MFuncResetAllFast),
		stFeedGroupTable	:= Table,
		nFilledRows			=> FilledRows,
		bError				=> ,
		nErrorId			=> );

	IF TblPrep.bError 
	THEN
		Error												:= TRUE;
		ErrorText											:= CONCAT('MFuncResetAllFast - JobNo. :',UDINT_TO_STRING(MFuncResetAllFast.nDisplayIndex));
		ErrorId												:= TblPrep.nErrorId;
	ELSE
		insertMFuncResetAllFast								:= TRUE;
	END_IF
END_METHOD

METHOD insertPathDynamics : BOOL //Return value = TRUE if executed succesful
VAR_IN_OUT
	Table													: ST_NciFeedGroupTable;
END_VAR
	TblPrep(
		nEntryType			:= PathDynamics.nEntryType,
		pEntry				:= ADR(PathDynamics),
		stFeedGroupTable	:= Table,
		nFilledRows			=> FilledRows,
		bError				=> ,
		nErrorId			=> );

	IF TblPrep.bError 
	THEN
		Error												:= TRUE;
		ErrorText											:= CONCAT('PathDynamics - JobNo. :',UDINT_TO_STRING(PathDynamics.nDisplayIndex));
		ErrorId												:= TblPrep.nErrorId;
	ELSE
		insertPathDynamics									:= TRUE;
	END_IF
END_METHOD

METHOD insertSetCoordinateSystem : bool //Return value = TRUE if executed succesful
VAR_IN_OUT
	Table													: ST_NciFeedGroupTable;
END_VAR
	TblPrep(
		nEntryType			:= SetCoordinateSystem.nEntryType,
		pEntry				:= ADR(SetCoordinateSystem),
		stFeedGroupTable	:= Table,
		nFilledRows			=> FilledRows,
		bError				=> ,
		nErrorId			=> );

	IF TblPrep.bError 
	THEN
		Error												:= TRUE;
		ErrorText											:= CONCAT('SetCoordinateSystem - JobNo. :',UDINT_TO_STRING(SetCoordinateSystem.nDisplayIndex));
		ErrorId												:= TblPrep.nErrorId;
	ELSE
		insertSetCoordinateSystem							:= TRUE;
	END_IF
END_METHOD

METHOD insertSParam : bool //Return value = TRUE if executed succesful
VAR_IN_OUT
	Table													: ST_NciFeedGroupTable;
END_VAR
	TblPrep(
		nEntryType			:= SParam.nEntryType,
		pEntry				:= ADR(SParam),
		stFeedGroupTable	:= Table,
		nFilledRows			=> FilledRows,
		bError				=> ,
		nErrorId			=> );

	IF TblPrep.bError 
	THEN
		Error												:= TRUE;
		ErrorText											:= CONCAT('SParam - JobNo. :',UDINT_TO_STRING(SParam.nDisplayIndex));
		ErrorId												:= TblPrep.nErrorId;
	ELSE
		insertSParam										:= TRUE;
	END_IF
END_METHOD

METHOD insertTangFollowingDesc : booL //Return value = TRUE if executed succesful
VAR_IN_OUT
	Table													: ST_NciFeedGroupTable;
END_VAR
	TblPrep(
		nEntryType			:= TangentialFollowingDesc.nEntryType,
		pEntry				:= ADR(TangentialFollowingDesc),
		stFeedGroupTable	:= Table,
		nFilledRows			=> FilledRows,
		bError				=> ,
		nErrorId			=> );

	IF TblPrep.bError 
	THEN
		Error												:= TRUE;
		ErrorText											:= CONCAT('TangentialFollowingDesc - JobNo. :','~');
		ErrorId												:= TblPrep.nErrorId;
	ELSE
		insertTangFollowingDesc								:= TRUE;
	END_IF
END_METHOD

METHOD insertTParam : bool //Return value = TRUE if executed succesful
VAR_IN_OUT
	Table													: ST_NciFeedGroupTable;
END_VAR
	TblPrep(
		nEntryType			:= TParam.nEntryType,
		pEntry				:= ADR(TParam),
		stFeedGroupTable	:= Table,
		nFilledRows			=> FilledRows,
		bError				=> ,
		nErrorId			=> );

	IF TblPrep.bError 
	THEN
		Error												:= TRUE;
		ErrorText											:= CONCAT('TParam - JobNo. :',UDINT_TO_STRING(TParam.nDisplayIndex));
		ErrorId												:= TblPrep.nErrorId;
	ELSE
		insertTParam										:= TRUE;
	END_IF
END_METHOD

METHOD insertVertexSmoothing : BOOL //Return value = TRUE if executed succesful
VAR_IN_OUT
	Table													: ST_NciFeedGroupTable;
END_VAR
	TblPrep(
		nEntryType			:= VertexSmoothing.nEntryType,
		pEntry				:= ADR(VertexSmoothing),
		stFeedGroupTable	:= Table,
		nFilledRows			=> FilledRows,
		bError				=> ,
		nErrorId			=> );

	IF TblPrep.bError 
	THEN
		Error												:= TRUE;
		ErrorText											:= CONCAT('VertexSmoothing - JobNo. :',UDINT_TO_STRING(VertexSmoothing.nDisplayIndex));
		ErrorId												:= TblPrep.nErrorId;
	ELSE
		insertVertexSmoothing								:= TRUE;
	END_IF
END_METHOD

METHOD reset : BOOL  //Return value = TRUE if execution finished
VAR_IN_OUT
	Table													: ST_NciFeedGroupTable;
END_VAR
TblPrep(
	nEntryType			:= ,
	pEntry				:= ,
	bResetTable			:= TRUE,
	bResetAll			:= TRUE,
	stFeedGroupTable	:= Table,
	nFilledRows			=> FilledRows,
	bError				=> ,
	nErrorId			=> );

TblPrep.bResetTable											:= FALSE;
TblPrep.bResetAll											:= FALSE;
Error														:= FALSE;
ErrorText													:= '';
ErrorId														:= 0;
Reset														:= TRUE;
END_METHOD

END_FUNCTION_BLOCK

// POUs/Motion/TF511x-KIN/03_DUTs/Trafo/UCS
{attribute 'hide'}
FUNCTION_BLOCK UCS
VAR_INPUT
	oid														:	UDINT := 0;		//Object identifier
	vTranslation 											:	VECTOR;
 	vRotation 												:	VECTOR;
	Valid													:	BOOL := FALSE;
END_VAR
VAR_OUTPUT
END_VAR
VAR
END_VAR

METHOD delete : BOOL
VAR_INPUT
END_VAR
MEMSET(ADR(vTranslation),0,SIZEOF(vTranslation));
MEMSET(ADR(VRotation),0,SIZEOF(VRotation));
oid 													:= 0;
delete	:= TRUE;
END_METHOD

END_FUNCTION_BLOCK

// POUs/Motion/TF5100-NCI/02_Options/RParameter/NCiReadWriteRParam
// To Start read or write, set inpult values and call action read/write. Busy and Done show the status of the operation
FUNCTION_BLOCK NCiReadWriteRParam EXTENDS FbBase
VAR_OUTPUT CONSTANT
	FNC_READ												:	INT := 0;
	FNC_WRITE												:	INT := 1;
END_VAR         											
VAR_INPUT       											
	Fnc														:	INT (FNC_READ..FNC_WRITE) := FNC_READ;
  	pAddr    												: 	PVOID; //Address of parameter destination variable
   	Index   												: 	DINT; //Index to parameter to read
   	Count   												: 	DINT; //
	rNCIRef													:	REFERENCE TO NCI_REF := 0;
END_VAR
VAR_OUTPUT
END_VAR
VAR
(* cache *******************************************************************)
	MemFnc													:	INT := -1;

(* trigger *****************************************************************)

(* function-block instances	************************************************)
	ItpReadRParamsEx										:	ItpReadRParamsEx := (tTimeout := DEFAULT_ADS_TIMEOUT);
	ItpWriteRParamsEx										:	ItpWriteRParamsEx := (tTimeout := DEFAULT_ADS_TIMEOUT);

END_VAR

	(* Read/Write Nci group R parameter													*)
	(************************************************************************************)

(* Execute ******************************************************************************)
	rtExecute(CLK := Execute);
	IF rtExecute.Q
		AND MemFnc < 0
	THEN
		MemFnc 												:= SEL(Fnc = FNC_WRITE, FNC_READ , FNC_WRITE) ;
		Busy												:= TRUE;
		Done												:= FALSE;
		Error												:= FALSE;
		ErrorID												:= 0;
	END_IF

(* Call Method ***************************************************************************)
	CASE MemFnc OF
	FNC_READ:
		Read(Execute );

	FNC_WRITE:
		Write(Execute );

	-1:
		IF NOT Execute
		THEN
			Busy											:= FALSE;
			Done											:= FALSE;
			Error											:= FALSE;
			ErrorID											:= 0;
		END_IF                              				
	ELSE                                    				
		Busy												:= FALSE;
		Done												:= FALSE;
		Error												:= Execute;
		ErrorID												:= E_AdsErr.DEVICE_INVALIDPARM;
	END_CASE

(*************************************************************************************************)

METHOD PUBLIC read : BOOL //Return value = TRUE if busy
//required parameter
//pAddr
//Index
//Count
//rNCIRef
VAR_INPUT 
	Execute													:	BOOL;
END_VAR
	MemFnc 													:= FNC_READ;
	This^.Execute											:= Execute;
IF NOT __ISVALIDREF(rNCIRef) OR pAddr = 0 
THEN
	Busy													:= NOT Error;
	ErrorId													:= E_adsErr.DEVICE_INVALIDPARM;
	Error													:= TRUE;
	Done													:= FALSE;
	MemFnc													:= SEL(Execute , -1 ,MemFnc); 
	RETURN;
END_IF
	
	IF Execute
	THEN
		Error												:=	FALSE;
		ErrorId												:= 0;
		ItpReadRParamsEx.bExecute 							:= TRUE;
	ELSIF NOT ItpReadRParamsEx.bBusy    					
	THEN                                					
		Error												:=	FALSE;
		ErrorId												:= 0;
		ItpReadRParamsEx.bExecute 							:= FALSE;

	END_IF

	ItpReadRParamsEx(
		bExecute	:= ,
		pAddr		:= pAddr,
		nIndex		:= Index,
		nCount		:= Count,
		tTimeOut	:= ,
		sNciToPlc	:= rNCIRef.NciToPlc,
		bBusy		=> Busy,
		bErr		=> ,
		nErrId		=> );

	Done													:= NOT ItpReadRParamsEx.bBusy
																AND NOT ItpReadRParamsEx.bErr
																AND ItpReadRParamsEx.bExecute;
                                                        	
	IF NOT Busy                                         	
	THEN                                                	
		IF ItpReadRParamsEx.bExecute                    	
		THEN                                            	
			Error											:=	ItpReadRParamsEx.bErr;
			ErrorId											:= ItpReadRParamsEx.nErrId;
		END_IF                          					
		IF NOT Execute                  					
		THEN                            	            	
			MemFnc											:= -1;
			ItpReadRParamsEx(bExecute := FALSE , sNciToPlc:= rNCIRef.NciToPlc);
		END_IF
	END_IF
	
	read													:= Busy;
END_METHOD

METHOD PUBLIC write : BOOL //Return value = TRUE if busy
//required parameter
//pAddr
//Index
//Count
//rNCIRef
VAR_INPUT
	Execute													:	BOOL;
END_VAR
	MemFnc 													:= FNC_WRITE;
	THIS^.Execute											:= Execute;

IF NOT __ISVALIDREF(rNCIRef) OR pAddr = 0 
THEN
	Busy													:= NOT Error;
	ErrorId													:= E_adsErr.DEVICE_INVALIDPARM;
	Error													:= TRUE;
	Done													:= FALSE;
	MemFnc													:= SEL(Execute , -1 ,MemFnc); 
	RETURN;
END_IF

	IF Execute
	THEN
		Error												:=	FALSE;
		ErrorId												:= 0;
		ItpWriteRParamsEx.bExecute 							:= TRUE;
	ELSIF NOT ItpWriteRParamsEx.bBusy   					
	THEN                                					
		Error												:=	FALSE;
		ErrorId												:= 0;
		ItpWriteRParamsEx.bExecute 							:= FALSE;

	END_IF

	ItpWriteRParamsEx(
		bExecute	:= ,
		pAddr		:= pAddr,
		nIndex		:= Index,
		nCount		:= Count,
		tTimeOut	:= ,
		sNciToPlc	:= rNCIRef.NciToPlc,
		bBusy		=> Busy,
		bErr		=> ,
		nErrId		=> );

	Done													:= NOT ItpWriteRParamsEx.bBusy
																AND NOT ItpWriteRParamsEx.bErr
																AND ItpWriteRParamsEx.bExecute;
                                        					
	IF NOT Busy
	THEN
		IF ItpWriteRParamsEx.bExecute
		THEN
			Error											:=	ItpWriteRParamsEx.bErr;
			ErrorId											:= ItpWriteRParamsEx.nErrId;
		END_IF                          					
		IF NOT Execute                  					
		THEN                            	
			MemFnc											:= -1;
			ItpWriteRParamsEx(bExecute := FALSE, sNciToPlc:= rNCIRef.NciToPlc);
		END_IF
	END_IF
	
	write													:= Busy;
END_METHOD

END_FUNCTION_BLOCK

// POUs/Motion/TF5100-NCI/NciChannel
{attribute 'no_check'}
FUNCTION_BLOCK NciChannel EXTENDS NCI_REF
VAR_INPUT
	Admin													:	NciAdmin;
	grp														:	NciGrp;
	Itp														:	NciItp;
	motion													:	NciMotion;
                        								   
	MFnc													: 	NciMFnc;
	RPara													:	NciReadWriteRParam;
                        								      
	Event													:	NciEventHandling;
                        	
END_VAR                 	
VAR_OUTPUT              	
	ErrHdl													:	ERROR_HDL;
END_VAR
VAR
END_VAR

	(* NCI Control											*)
	(********************************************************)

(********************************************************************************)
(* error event ctrl																*)
(********************************************************************************)
	Event(
		Enable			:= ,
		ConfirmTrig		:= NOT Errhdl.flag AND Event.Status.31 OR Admin.ResetAdmin,
		Name			:= ErrHdl.fnc,
		SourceId		:= (* Default *) ,
		rNci			:= THIS^,
		ErrorId			:= TO_UDINT(ErrHdl.Id),
		Status			=> );
		
	(* Reset FB errors by reset flag *)
	(* currently not in use, call _Resetting via state machine to reset Fb errors by setting Execute to FALSE 
	IF Admin.Reset
	THEN
		grp.Execute											:= grp.Execute AND NOT grp.Error;
		itp.Execute											:= itp.Execute AND NOT itp.Error;
		Motion.Execute										:= Motion.Execute AND NOT Motion.Error;
		RPara.Execute										:= RPara.Execute AND NOT RPara.Error;
	END_IF
	*)
	
(********************************************************************************)
(* work admin ctrl																*)
(********************************************************************************)
	admin(
		ResetAdmin					:= ,
		Enable					:= ,
		EStop					:= ,
		SingleBlockMode			:= , 
		InSingleBlockTrigNext	:= , 
		GrpCnfg					:= ,
		Override				:= ,
		SpindleOvr				:= ,	
		rNCIRef					:= THIS^,
		InGroup					=> ,
		Busy					=> ,
		Done					=> ,
		Error					=> ,
		ErrorID					=> ,
		ErrorText				=> );

(********************************************************************************)
(* work group ctrl																*)
(********************************************************************************)
	grp(
		Execute				:= ,
		Fnc					:= ,
		XAxisId				:= ,
		YAxisId				:= ,
		ZAxisId				:= ,
		Q1AxisId			:= ,
		Q2AxisId			:= ,
		Q3AxisId			:= ,
		Q4AxisId			:= ,
		Q5AxisId			:= ,
		AxisIndex			:= ,
		rNCIRef				:= THIS^, 
		Busy				=> ,
		Done				=> ,
		Error				=> ,
		ErrorID				=> ,
		ErrorText			=> );

(********************************************************************************)
(* work interpolation ctrl														*)
(********************************************************************************)
	Itp(
		Execute				:= ,
		Fnc					:= ,
		Prg					:= ,
		rTable				:= ,
		rNCIRef				:= THIS^,
		StartPrgAfterLoading:= , 
		LogFeederEntries	:= ,
		Busy				=> ,
		Done				=> ,
		Error				=> ,
		ErrorID				=> ,
		ErrorText			=> );


(********************************************************************************)
(* work motion ctrl																*)
(********************************************************************************)
	motion(
		Execute						:= ,
		Fnc							:= ,
		rNCIRef						:= THIS^,
		FNC_ESTOP					=> ,
		FNC_STEP_ON					=> ,
		FNC_ENABLE_FEEDER_BACKUP	=> ,
		FNC_DISABLE_FEEDER_BACKUP	=> ,
		FNC_RETRACE_FWD				=> ,
		FNC_RETRACE_BWD				=> ,
		Busy						=> ,
		Done						=> ,
		Error						=> ,
		ErrorId						=> ,
		ErrorText					=> );

(********************************************************************************)
(* work R rarameter ctrl														*)
(********************************************************************************)
	RPara(
		Execute						:= ,
		Fnc							:= ,
		pAddr						:= ,
		Index						:= ,
		Count						:= ,
		rNCIRef						:= THIS^,
		Done						=> ,
		Busy						=> ,
		Error						=> ,
		ErrorId						=> );

(********************************************************************************)
(* work M function  ctrl														*)
(********************************************************************************)
	MFnc(
		ConfirmHsk					:= ,
		FastMFuncReset				:= ,
		FastMFuncNo					:= ,
		rNCIRef						:= THIS^);

(********************************************************************************)
(* collect errors																*)
(********************************************************************************)
	IF Admin.Error
	THEN
		ErrHdl.flag											:= Admin.Error;
		ErrHdl.id											:= UDINT_TO_DINT(Admin.ErrorID);
		ErrHdl.fnc											:= 'NciAdmin';
		ErrHdl.text											:= Admin.ErrorText;
                        									
	ELSIF grp.Error     									
	THEN                									
		ErrHdl.flag											:= grp.Error;
		ErrHdl.id											:= UDINT_TO_DINT(grp.ErrorID);
		ErrHdl.fnc											:= 'NciGrp';
		ErrHdl.text											:= grp.ErrorText;
                        									
	ELSIF itp.Error     									
	THEN                									
		ErrHdl.flag											:= Itp.Error;
		ErrHdl.id											:= UDINT_TO_DINT(Itp.ErrorID);
		ErrHdl.fnc											:= 'NciItp';
		ErrHdl.text											:= Itp.ErrorText;
                        									
	ELSIF motion.Error  									
	THEN                									
		ErrHdl.flag											:= motion.Error;
		ErrHdl.id											:= UDINT_TO_DINT(motion.ErrorID);
		ErrHdl.fnc											:= 'NciMotion';
		ErrHdl.text											:= motion.ErrorText;
		
	ELSIF RPara.Error  									
	THEN                									
		ErrHdl.flag											:= RPara.Error;
		ErrHdl.id											:= UDINT_TO_DINT(RPara.ErrorID);
		ErrHdl.fnc											:= 'RPara';
		ErrHdl.text											:= CONCAT('Error RPara id: ',  UDINT_TO_STRING(RPara.Errorid));
	ELSE
		ErrHdl.Reset();
	END_IF
(******************************************************************************)

METHOD PUBLIC noAction : BOOL
VAR_INPUT
END_VAR
grp.Execute													:= FALSE;
itp.Execute													:= FALSE;
Motion.Execute												:= FALSE;
RPara.Execute												:= FALSE;

NoAction 													:= NOT Grp.Busy and not Itp.Busy and not Motion.Busy and not RPara.Busy;
END_METHOD

METHOD reset : Bool
VAR_INPUT
END_VAR
NoAction();
reset 			:= ErrHdl.flag OR Admin.reset(FALSE);
Event.confirm();
END_METHOD

END_FUNCTION_BLOCK

// POUs/Motion/TF511x-KIN/01_Main/KIN_REF
//Kinematic group ref - call ReadStatus cyclic
FUNCTION_BLOCK KIN_REF
VAR_INPUT
	PlcToNci										AT %Q*	:	PLCTONC_NCICHANNEL_REF;
END_VAR                     						
VAR_OUTPUT                  						
	NciToPlc										AT %I*	:	NCTOPLC_NCICHANNEL_REF;
                            						
	ChnOperationState										:	E_KINSTATUS := 0;
	CartesianModeON											:	BOOL := FALSE;
	                                					
(* ChnState ***************************)
	IsKinematicChn											:	BOOL := FALSE;
	                                					
	AxList													: ST_KinAxes;
END_VAR
VAR
END_VAR

;

METHOD PUBLIC readStatus : booL;
VAR_INPUT
END_VAR
(* Kin Channel State *********************************************************)
	F_KinGetAcsMcsAxisIds(AxList,NciToPlc);
	
	ChnOperationState 										:= TO_INT(F_KinGetChnOperationState(NciToPlc));

	CartesianModeON											:= NciToPlc.AcsAxisIDs[0] <> 0 AND NciToPlc.AcsAxisIDs[1] <> 0;
	
	IsKinematicChn											:= NciToPlc.ChnState.1;

	readStatus												:= TRUE;
(*****************************************************************************)
END_METHOD

END_FUNCTION_BLOCK

// POUs/Motion/TF511x-KIN/01_Main/KinAdmin
//Kinematic group administration - Enable/Disable/Reset group
//based on TF511x - Tc2_NcKinematicTransformation
//ACS - Axis coordinate system => Robot motors M1-Mx 
//MCS - Machine coordinate system >= Cartesian Axis X,Y,Z,Rx,Ry,Rz (A,B,C) 
FUNCTION_BLOCK KinAdmin
VAR_INPUT
	ResetTrig												:	BOOL := FALSE;
	Enable													:	BOOL := FALSE; (* TRUE = Build Group , FALSE = Reconfig Group *)
	Override												:	LREAL	:= 0.0;
	ItpChannelId 											: 	UDINT := 0; (* Bei 0 wirtd der ITP Kanal nicht resetet *)
	AxesList												: 	ST_KinAxes;
	rKINRef													:	REFERENCE TO KIN_REF := 0;
END_VAR
VAR_IN_OUT
END_VAR
VAR_OUTPUT
	Busy													:	BOOL;
	Done													:	BOOL;
	Error													:	BOOL;
{attribute 'displaymode':='hex'}
	ErrorId													:	UDINT;
	ErrorText												:	STRING(40);
END_VAR
VAR
(* cache **************************************************************************)
	MemDone													:	BOOL;
	MemFnc													:	INT := 1;
	                        								
(* MC-functonblock instances *******************************************************)
	ResetKinGroup											: 	FB_KinResetGroup ;
	ConfigKinGroup											:	FB_KinConfigGroup  ;

(* Dummy Speicher **********************************************************)
	OK 														: BOOL;
END_VAR

	(* Kinematic group administration										*)
	(************************************************************************)

(* aborting function-block call if pointer is not valid ****************************************)
IF NOT __ISVALIDREF(rKINRef) 
THEN
	Busy													:= NOT Error;
	ErrorId													:= E_AdsErr.DEVICE_INVALIDPARM;
	Error													:= TRUE;
	Done													:= FALSE;
	ErrorText												:= 'Reference to rKINRef invalid (0)';
	RETURN;
END_IF

(* reading axis-status from NCtoPLC-channel ***************************************************)
	rKINRef.readStatus();

(* accepting setvalue-barrier e.g. for hardware limit switch **********************************)
	rKINRef.PlcToNci.ChnAxesOvr 							:= LREAL_TO_DWORD(LIMIT(0.0,Override,100.0) * 10000.0 );

(* ctrl programm ******************************************************************************)
	ConfigKinGroup.bExecute									:=	NOT ConfigKinGroup.bBusy
																AND(
																Enable
																AND NOT ConfigKinGroup.bCartesianMode
																OR
																NOT Enable
																AND ConfigKinGroup.bCartesianMode);

	IF ConfigKinGroup.bExecute
	THEN
		ConfigKinGroup.bCartesianMode						:= Enable;
	END_IF

	ConfigKinGroup(
		bExecute		:= ,
		bCartesianMode	:= ,
		stAxesList		:= AxesList,
		stKinRefIn		:= rKinRef.NciToPlc,
		bBusy			=> ,
		bDone			=> ,
		bError			=> ,
		nErrorId		=> );

(* Reset Grp ****************************************************************)
	IF Memfnc < 0
	THEN
		IF ResetTrig
		THEN
			reset(Execute:= TRUE);
			MemFnc											:= 1;
		END_IF
	ELSIF NOT reset(Execute:= ResetTrig)
	THEN
		MemFnc												:= -1;
	END_IF

(******************************************************************************)
(* Ctrl Status 																					*)
(******************************************************************************)
	Busy						:= ResetKinGroup.bBusy OR ConfigKinGroup.bBusy;
	
	IF Busy
	THEN
		Error												:= FALSE;
		ErrorId												:= 0;
		ErrorText											:= '';
	ELSIF ConfigKinGroup.bError
	THEN
		Error												:= TRUE;
		ErrorId												:= ConfigKinGroup.nErrorID;
		ErrorText											:= CONCAT('ConfigKinGroup ErrorId: ', UDINT_TO_STRING(Errorid));
	ELSIF ResetKinGroup.bExecute
		AND ResetKinGroup.bError
	THEN
		Error												:= TRUE;
		ErrorId												:= ResetKinGroup.nErrorID;
		ErrorText											:= CONCAT('ResetKinGroup ErrorId: ', UDINT_TO_STRING(Errorid));
	ELSIF rKINRef.NciToPlc.ErrorCode <> 0
	THEN
		Error												:= TRUE;
		ErrorId												:= rKINRef.NciToPlc.ErrorCode;
		ErrorText											:= CONCAT('KIN Grp ErrorId: ', UDINT_TO_STRING(Errorid));
	ELSE
		Error												:= FALSE;
		ErrorId												:= 0;
		ErrorText											:= '';
	END_IF

	IF ResetKinGroup.bDone
		OR ConfigKinGroup.bDone
	THEN
		MemDone												:= TRUE;
	END_IF

	Done													:= NOT Busy AND MemDone;

	IF done
	THEN
		MemDone												:= FALSE;
	END_IF

(**************************************************************************************************)

METHOD PUBLIC reset : BOOL //Return value = TRUE if busy
//required parameter
//rKinRef
//ItpChannelId
//AxesList
VAR_INPUT
	Execute													:	BOOL;
END_VAR
IF NOT __ISVALIDREF(rKINRef) THEN
	Busy													:= NOT Error;
	ErrorId													:=E_AdsErr.DEVICE_INVALIDPARM;
	Error													:= TRUE;
	Done													:= FALSE;
	ErrorText												:= 'Reference to rKINRef  invalid (0)';
	RETURN;
END_IF

	IF Execute
	THEN
		Error												:=	FALSE;
		ErrorId												:= 0;
		ResetKinGroup.bExecute 								:= rKinRef.NciToPlc.ErrorCode <> 0;
	ELSIF NOT ResetKinGroup.bBusy
	THEN
		Error												:=	FALSE;
		ErrorId												:= 0;
		ResetKinGroup.bExecute 								:= FALSE;

	END_IF

	ResetKinGroup(
		bExecute		:= ,
		nItpChannelId	:= ItpChannelId,
		stKinRefIn		:= rKinRef.NciToPlc,
		stAxesList		:= AxesList,
		bBusy			=> Busy,
		bDone			=> ,
		bError			=> ,
		nErrorId		=> );

	Done													:= NOT ResetKinGroup.bBusy
																AND NOT ResetKinGroup.bError
																AND ResetKinGroup.bExecute;

	IF NOT Busy
	THEN
		IF ResetKinGroup.bExecute
		THEN
			Error											:=	ResetKinGroup.bError;
			ErrorId											:= ResetKinGroup.nErrorId;
			ErrorText										:= SEL(Error , '' ,  CONCAT('Error ResetKinGroup id: ',  UDINT_TO_STRING(Errorid)));
		END_IF
		IF NOT Execute
		THEN
			MemFnc											:= -1 ;
			ResetKinGroup(	bExecute := FALSE, 
							stKinRefIn := rKinRef.NciToPlc, 
							stAxesList := AxesList);
		END_IF
	END_IF
	
	reset													:= Busy;
END_METHOD

END_FUNCTION_BLOCK

// POUs/Motion/TF511x-KIN/02_Options/KinLockUnlockTrafoParam
//Lock or Unlock kinematic group parameter
FUNCTION_BLOCK KinLockUnlockTrafoParam
VAR_INPUT
	Execute													:	BOOL	:= FALSE;
	Lock													:	BOOL 	:= TRUE;
   	oidTrafo												:	UDINT;
END_VAR                     								
VAR_OUTPUT                  								
	Busy													:	BOOL	:= FALSE;
	Done													:	BOOL	:= FALSE;
	Error													:	BOOL	:= FALSE;
	ErrorId													:	UDINT	:= 0;
END_VAR                     								
VAR                         	
	State													:	UDINT	:= 0;
	ADSWRITE												:	ADSWRITE;
END_VAR

CASE State OF
0:
	Done													:= FALSE;
	Error													:= FALSE;
	ErrorId													:= 0;
	Busy 													:= FALSE;
	
	IF Execute THEN
		AdsWrite(WRITE := FALSE);
		AdsWrite(
			NETID		:='',
			PORT		:= 10,
			IDXGRP		:=oidTrafo,
			IDXOFFS		:=SEL(Lock, 16#05030210, 16#0503020F),
			LEN			:= 0,
			SRCADDR		:=0 ,
			WRITE		:= TRUE,
			TMOUT		:= DEFAULT_ADS_TIMEOUT,
			BUSY		=> ,
			ERR			=> ,
			ERRID		=> );

		Busy												:= TRUE;
		State												:= 10;
	END_IF
10:
	AdsWrite(
		TMOUT	:= DEFAULT_ADS_TIMEOUT,
		BUSY	=>,
		ERR		=>Error,
		ERRID	=>ErrorId);
		
	IF NOT AdsWrite.BUSY 
	THEN
		IF NOT AdsWrite.ERR 
		THEN
			Done											:= TRUE;
		END_IF
		IF NOT Execute THEN
			State											:= 0;
		ELSE
			State											:= 20;
		END_IF
		AdsWrite(WRITE:=FALSE);
	END_IF
20:
	Busy													:= FALSE;
	IF NOT Execute THEN
		State												:= 0;
	END_IF

END_CASE

END_FUNCTION_BLOCK

// POUs/Motion/TF511x-KIN/02_Options/KinWriteToolTrafoParam
{attribute 'hide'}
(*==============================================================================*)
(* Name:			KIN_WriteToolTrafoParam							  	 		*)
(* Desc:			THIS IS NOT A RELEASED IMPLEMENTATION AND    				*)
(*  	           	SUBJECT TO CHANGE                            				*)
(*     			 															    *)
(* Author:	 	DS																*)
(* Date:							     										*)
(*==============================================================================*)
FUNCTION_BLOCK KinWriteToolTrafoParam
VAR_INPUT
	Execute													:	BOOL	:= FALSE;
   	oidTrafo												:	UDINT;
	ToolX													:	LREAL := 0.0;
	ToolY													:	LREAL := 0.0;
	ToolZ													:	LREAL := 0.0;
END_VAR                     								
VAR_OUTPUT                  								
	Busy													:	BOOL	:= FALSE;
	Done													:	BOOL	:= FALSE;
	Error													:	BOOL	:= FALSE;
	ErrorId													:	UDINT	:= 0;
END_VAR
VAR
	State													:	UDINT	:= 0;
	ADSWRITE												:ADSWRITE;
END_VAR

CASE State OF
0:
	Done													:= FALSE;
	Busy 													:= FALSE;
	Error													:= FALSE;
	ErrorId													:= 0;
	IF Execute 
	THEN
		AdsWrite(WRITE := FALSE);
		AdsWrite(
			NETID	:='',
			PORT	:= 10,
			IDXGRP	:=oidTrafo,
			IDXOFFS	:=SEL(FALSE (* Lock *), 16#05030210, 16#0503020F),
			LEN		:= 0,
			SRCADDR	:=0 ,
			WRITE	:= TRUE,
			TMOUT	:= DEFAULT_ADS_TIMEOUT,
			BUSY	=> ,
			ERR		=> ,
			ERRID	=> );

		Busy												:= TRUE;
		State												:= 1;
	END_IF

1:
	AdsWrite(
		TMOUT	:= DEFAULT_ADS_TIMEOUT,
		BUSY	=>,
		ERR		=>Error,
		ERRID	=>ErrorId);
		
	IF NOT AdsWrite.BUSY 
	THEN
		AdsWrite(WRITE:=FALSE);
			
		IF NOT AdsWrite.ERR 
		THEN
			AdsWrite( (* Write Tool X *)
				NETID	:= '',
				PORT	:= 10,
				IDXGRP	:= oidTrafo, 				(*OID 	Tool trafo*)
				IDXOFFS	:= 16#05010020, 			(*PTCID	Tool Trafo Parameter*)
				LEN		:= SIZEOF(ToolX),
				SRCADDR	:= ADR(ToolX),
				TMOUT	:= DEFAULT_ADS_TIMEOUT,
				WRITE 	:= TRUE,
				BUSY	=> ,
				ERR		=> ,
				ERRID	=> );
	

			State											:= 10;
		ELSE
			IF NOT Execute
			THEN
				State										:= 0;
			ELSE
				State										:= 99;
			END_IF
		END_IF
	END_IF

10:
	AdsWrite(
		TMOUT	:= DEFAULT_ADS_TIMEOUT,
		BUSY	=>,
		ERR		=>Error,
		ERRID	=>ErrorId);
		
	IF NOT AdsWrite.BUSY 
	THEN
		AdsWrite(WRITE:=FALSE);
		
		IF NOT AdsWrite.ERR 
		THEN
			AdsWrite( 								(* Write Tool Y *)
				NETID	:= '',
				PORT	:= 10,
				IDXGRP	:= oidTrafo, 				(*OID 	Tool trafo*)
				IDXOFFS	:= 16#05010021, 			(*PTCID	Tool Trafo Parameter*)
				LEN		:= SIZEOF(ToolY),
				SRCADDR	:= ADR(ToolY),
				TMOUT	:= DEFAULT_ADS_TIMEOUT,
				WRITE	:= TRUE,
				BUSY	=> ,
				ERR		=> ,
				ERRID	=> );

			State											:= 20;
		ELSE
			State											:= 90;
		END_IF
	END_IF

20:
	AdsWrite(
		TMOUT	:= DEFAULT_ADS_TIMEOUT,
		BUSY	=>,
		ERR		=>Error,
		ERRID	=>ErrorId);

	IF NOT AdsWrite.BUSY 
	THEN
		AdsWrite(WRITE:=FALSE);
		
	IF NOT AdsWrite.ERR 
	THEN
			AdsWrite( 								(* Write Tool Z *)
				NETID	:= '',
				PORT	:= 10,
				IDXGRP	:= oidTrafo, 				(*OID 	Tool trafo*)
				IDXOFFS	:= 16#05010022, 			(*PTCID	Tool Trafo Parameter*)
				LEN		:= SIZEOF(ToolZ),
				SRCADDR	:= ADR(ToolZ),
				TMOUT	:= DEFAULT_ADS_TIMEOUT,
				WRITE 	:= TRUE,
				BUSY	=> ,
				ERR		=> ,
				ERRID	=> );

			State											:= 60;
		ELSE            									
			State											:= 90;
		END_IF
	END_IF

60:
	AdsWrite(
		TMOUT	:= DEFAULT_ADS_TIMEOUT,
		BUSY	=>,
		ERR		=>Error,
		ERRID	=>ErrorId);

	IF NOT AdsWrite.BUSY 
	THEN
		State												:= 90;
		AdsWrite(WRITE:=FALSE);
	END_IF


90: (* Start Lock-Param *)
	AdsWrite(
		NETID	:='',
		PORT	:= 10,
		IDXGRP	:=oidTrafo,
		IDXOFFS	:=SEL(TRUE (* Lock *), 16#05030210, 16#0503020F),
		LEN		:= 0,
		SRCADDR	:=0 ,
		WRITE	:= TRUE,
		TMOUT	:= DEFAULT_ADS_TIMEOUT,
		BUSY	=> ,
		ERR		=> ,
		ERRID	=> );

	State													:= 91;

91:
	AdsWrite(
		TMOUT	:= DEFAULT_ADS_TIMEOUT,
		BUSY	=>,
		ERR		=>,
		ERRID	=>);

	IF NOT AdsWrite.BUSY 
	THEN
		Busy 												:= FALSE;
		IF NOT AdsWrite.ERR 
		THEN
			Done											:= NOT Error;
		ELSIF NOT Error
		THEN
			Error 											:= AdsWrite.ERR;
			ErrorId 										:= AdsWrite.ERRID;
		END_IF
		IF NOT Execute 
		THEN
			State											:= 0;
		ELSE        										
			State											:= 99;
		END_IF
		AdsWrite(WRITE:=FALSE);
	END_IF

99:
	Busy													:= FALSE;
	IF NOT Execute THEN
		State												:= 0;
	END_IF

END_CASE

END_FUNCTION_BLOCK

// POUs/Motion/TF511x-KIN/02_Options/KinWriteUCSTrafoParam
{attribute 'hide'}
(*==============================================================================*)
(* Name:			KIN_WriteUCSTrafoParam							  	 		*)
(* Desc:			THIS IS NOT A RELEASED IMPLEMENTATION AND    				*)
(*  	           	SUBJECT TO CHANGE                            				*)
(*     			 															    *)
(* Author:	 	DS																*)
(* Date:							     										*)
(*==============================================================================*)
FUNCTION_BLOCK KinWriteUCSTrafoParam
VAR_INPUT
	Execute													:	BOOL	:= FALSE;
   oidTrafo													:	UDINT;
	vTranslation 											:	VECTOR;
 	vRotation 												:	VECTOR;
END_VAR
VAR_OUTPUT
	Busy													:	BOOL	:= FALSE;
	Done													:	BOOL	:= FALSE;
	Error													:	BOOL	:= FALSE;
	ErrorId													:	UDINT	:= 0;
END_VAR
VAR
	State													:	UDINT	:= 0;
	ADSWRITE												:ADSWRITE;
END_VAR

CASE State OF
0:
	Done													:= FALSE;
	Busy													:= FALSE;
	Error													:= FALSE;
	ErrorId													:= 0;
	IF Execute 
	THEN
		AdsWrite(WRITE := FALSE);
		AdsWrite(
			NETID	:='',
			PORT	:= 10,
			IDXGRP	:=oidTrafo,
			IDXOFFS	:=SEL(FALSE (* Lock *), 16#05030210, 16#0503020F),
			LEN		:= 0,
			SRCADDR	:=0 ,
			WRITE	:= TRUE,
			TMOUT	:= DEFAULT_ADS_TIMEOUT,
			BUSY	=> ,
			ERR		=> ,
			ERRID	=> );

		Busy												:= TRUE;
		State												:= 1;
	END_IF

1: (* Start Translation X *)
	AdsWrite(
		TMOUT	:= DEFAULT_ADS_TIMEOUT,
		BUSY	=>,
		ERR		=>Error,
		ERRID	=>ErrorId);
		
	IF NOT AdsWrite.BUSY 
	THEN
		AdsWrite(WRITE:=FALSE);
		IF NOT AdsWrite.ERR 
		THEN
			AdsWrite(
				NETID	:= '',
				PORT	:= 10,
				IDXGRP	:= oidTrafo,
				IDXOFFS	:= 16#05010020,
				LEN		:= SIZEOF(vTranslation.m[1]),
				SRCADDR	:= ADR(vTranslation.m[1]),
				TMOUT	:= DEFAULT_ADS_TIMEOUT,
				WRITE 	:= TRUE,
				BUSY	=> ,
				ERR		=> ,
				ERRID	=> );

			State											:= 10;
		ELSE (* Error unlock Param *)
			IF NOT Execute 
			THEN
				State										:= 0;
			ELSE
				State										:= 99;
			END_IF
		END_IF
	END_IF

10: (* Translation Y *)
	AdsWrite(
		TMOUT	:= DEFAULT_ADS_TIMEOUT,
		BUSY	=>,
		ERR		=>Error,
		ERRID	=>ErrorId);
		
	IF NOT AdsWrite.BUSY 
	THEN
		AdsWrite(WRITE:=FALSE);
		
		IF NOT AdsWrite.ERR 
		THEN
			AdsWrite(
				NETID	:= '',
				PORT	:= 10,
				IDXGRP	:= oidTrafo,
				IDXOFFS	:= 16#05010021,
				LEN		:= SIZEOF(vTranslation.m[2]),
				SRCADDR	:= ADR(vTranslation.m[2]),
				TMOUT	:= DEFAULT_ADS_TIMEOUT,
				WRITE 	:= TRUE,
				BUSY	=> ,
				ERR		=> ,
				ERRID	=> );

			State											:= 20;
		ELSE            									
			State											:= 90;
		END_IF

	END_IF

20: (* Translation Z *)
	AdsWrite(
		TMOUT	:= DEFAULT_ADS_TIMEOUT,
		BUSY	=>,
		ERR		=>Error,
		ERRID	=>ErrorId);

	IF NOT AdsWrite.BUSY 
	THEN
		AdsWrite(WRITE:=FALSE);
		IF NOT AdsWrite.ERR 
		THEN
			AdsWrite(
				NETID	:= '',
				PORT	:= 10,
				IDXGRP	:= oidTrafo,
				IDXOFFS	:= 16#05010022,
				LEN		:= SIZEOF(vTranslation.m[3]),
				SRCADDR	:= ADR(vTranslation.m[3]),
				TMOUT	:= DEFAULT_ADS_TIMEOUT,
				WRITE 	:= TRUE,
				BUSY	=> ,
				ERR		=> ,
				ERRID	=> );

			State											:= 30;
		ELSE
			State											:= 90;
		END_IF

	END_IF

30: (* Roation X *)
	AdsWrite(
		TMOUT	:= DEFAULT_ADS_TIMEOUT,
		BUSY	=>,
		ERR		=>Error,
		ERRID	=>ErrorId);

	IF NOT AdsWrite.BUSY 
	THEN
		AdsWrite(WRITE:=FALSE);
		IF NOT AdsWrite.ERR 
		THEN
			AdsWrite(
				NETID	:= '',
				PORT	:= 10,
				IDXGRP	:= oidTrafo,
				IDXOFFS	:= 16#05010060,
				LEN		:= SIZEOF(VRotation.m[1]),
				SRCADDR	:= ADR(VRotation.m[1]),
				TMOUT	:= DEFAULT_ADS_TIMEOUT,
				WRITE 	:= TRUE,
				BUSY	=> ,
				ERR		=> ,
				ERRID	=> );

			State											:= 40;
		ELSE
			State											:= 90;
		END_IF
	END_IF

40: (* Roation Y *)
	AdsWrite(
		TMOUT	:= DEFAULT_ADS_TIMEOUT,
		BUSY	=>,
		ERR		=>Error,
		ERRID	=>ErrorId);

	IF NOT AdsWrite.BUSY 
	THEN
		AdsWrite(WRITE:=FALSE);
		IF NOT AdsWrite.ERR 
		THEN
			AdsWrite(
				NETID	:= '',
				PORT	:= 10,
				IDXGRP	:= oidTrafo,
				IDXOFFS	:= 16#05010061,
				LEN		:= SIZEOF(VRotation.m[2]),
				SRCADDR	:= ADR(VRotation.m[2]),
				TMOUT	:= DEFAULT_ADS_TIMEOUT,
				WRITE 	:= TRUE,
				BUSY	=> ,
				ERR		=> ,
				ERRID	=> );
			State											:= 50;
		ELSE            									
			State											:= 90;
		END_IF

	END_IF

50: (* Roation Z *)
	AdsWrite(
		TMOUT	:= DEFAULT_ADS_TIMEOUT,
		BUSY	=>,
		ERR		=>Error,
		ERRID	=>ErrorId);

	IF NOT AdsWrite.BUSY 
	THEN
		AdsWrite(WRITE:=FALSE);
		IF NOT AdsWrite.ERR 
		THEN
			AdsWrite(
				NETID	:= '',
				PORT	:= 10,
				IDXGRP	:= oidTrafo,
				IDXOFFS	:= 16#05010062,
				LEN		:= SIZEOF(VRotation.m[3]),
				SRCADDR	:= ADR(VRotation.m[3]),
				TMOUT	:= DEFAULT_ADS_TIMEOUT,
				WRITE 	:= TRUE,
				BUSY	=> ,
				ERR		=> ,
				ERRID	=> );

			State											:= 60;
		ELSE            									
			State											:= 90;
		END_IF
	END_IF

60:
	AdsWrite(
		TMOUT	:= DEFAULT_ADS_TIMEOUT,
		BUSY	=>,
		ERR		=>Error,
		ERRID	=>ErrorId);

	IF NOT AdsWrite.BUSY 
	THEN
		State												:= 90;
		AdsWrite(WRITE:=FALSE);
	END_IF

90: (* Start Lock-Param *)
	AdsWrite(
		NETID	:='',
		PORT	:= 10,
		IDXGRP	:=oidTrafo,
		IDXOFFS	:=SEL(TRUE (* Lock *), 16#05030210, 16#0503020F),
		LEN		:= 0,
		SRCADDR	:=0 ,
		WRITE	:= TRUE,
		TMOUT	:= DEFAULT_ADS_TIMEOUT,
		BUSY	=> ,
		ERR		=> ,
		ERRID	=> );

	State													:= 91;

91:
	AdsWrite(
		TMOUT	:= DEFAULT_ADS_TIMEOUT,
		BUSY	=>,
		ERR		=>,
		ERRID	=>);

	IF NOT AdsWrite.BUSY 
	THEN
		Busy 												:= FALSE;
		IF NOT AdsWrite.ERR 
		THEN
			Done											:= NOT Error;
		ELSIF NOT Error
		THEN
			Error 											:= AdsWrite.ERR;
			ErrorId 										:= AdsWrite.ERRID;
		END_IF
		IF NOT Execute 
		THEN
			State											:= 0;
		ELSE        										
			State											:= 99;
		END_IF
		AdsWrite(WRITE:=FALSE);
	END_IF

99:
	Busy 													:= FALSE;
	IF NOT Execute 
	THEN
		State												:= 0;
	END_IF

END_CASE

END_FUNCTION_BLOCK

// POUs/Motion/TF511x-KIN/03_DUTs/Positions/KIN_POSITIONS
{attribute 'no_check'}
FUNCTION_BLOCK KIN_POSITIONS 
VAR_INPUT
	Valid													:	BOOL ;
	MCS														:	KIN_POSITIONS_MCS_DUT; //Values as union
END_VAR
VAR_OUTPUT
END_VAR
VAR
END_VAR

;

METHOD PUBLIC copy : BOOL //Return value = TRUE if execution finished
VAR_IN_OUT
	Source													:	KIN_POSITIONS;
END_VAR
	Valid													:= Source.Valid;
	MCS														:= Source.MCS;
	copy													:= TRUE;
END_METHOD

METHOD PUBLIC delete : BOOL //Return value = TRUE if execution finished - Valid bit will not change
VAR_INPUT
END_VAR
	MCS.A													:= 0.0;
	MCS.B													:= 0.0;
	MCS.C													:= 0.0;
	MCS.X													:= 0.0;
	MCS.Y													:= 0.0;
	MCS.Z													:= 0.0;
	MCS.Q1													:= 0.0;
	MCS.Q2													:= 0.0;
	
	delete													:= TRUE;
END_METHOD

METHOD PUBLIC isInPos : BOOL //Return value = TRUE if axes are within window of checkPos values
VAR_IN_OUT
	CheckPos												:	KIN_POSITIONS_MCS_DUT;
	Window													:	KIN_POSITIONS_MCS_DUT;
END_VAR             										
VAR CONSTANT        										
END_VAR
IsInPos 														:= IsInPosXYZ(CheckPos,Window) AND IsInPosABC(CheckPos,Window);
END_METHOD

METHOD PUBLIC isInPosABC : BOOL //Return value = TRUE if axes are within window of checkPos values
VAR_IN_OUT
	CheckPos												:	KIN_POSITIONS_MCS_DUT;
	Window													:	KIN_POSITIONS_MCS_DUT;
END_VAR                 									
VAR CONSTANT            									
END_VAR
isInPosABC												 	:= CAM(CheckPos.A, MCS.A ,Window.A)
																AND CAM(CheckPos.B, MCS.B ,Window.B)
																AND CAM(CheckPos.C, MCS.C ,Window.C);
END_METHOD

METHOD PUBLIC isInPosByAxisNo : BOOL //Return value = TRUE selected axis is within window of checkPos values
VAR_INPUT
	No					:	INT;
END_VAR
VAR_IN_OUT
	CheckPos			:	KIN_POSITIONS_MCS_DUT;
	Window				:	KIN_POSITIONS_MCS_DUT;
END_VAR
isInPosByAxisNo													:= (CAM(CheckPos.X, MCS.X ,Window.X) OR No <> 1)
																AND (CAM(CheckPos.Y, MCS.Y ,Window.Y) OR No <> 2)
																AND (CAM(CheckPos.Z, MCS.Z ,Window.Z) OR No <> 3)
																AND (CAM(CheckPos.A, MCS.A ,Window.A) OR No <> 4)
																AND (CAM(CheckPos.B, MCS.B ,Window.B) OR No <> 5)
																AND (CAM(CheckPos.C, MCS.C ,Window.C) OR No <> 6)
																AND (CAM(CheckPos.Q1, MCS.Q1 ,Window.Q1) OR No <> 7)
																AND (CAM(CheckPos.Q2, MCS.Q2 ,Window.Q2) OR No <> 8);
END_METHOD

METHOD PUBLIC isInPosExt : BOOL //Return value = TRUE if axes are within window of checkPos values
VAR_INPUT
{attribute 'displaymode':='binary'}
	Config													:	DWORD; //Select value to be checked by bis mask .0=X or A1, .1=Y or A2, .3=Y or A3.....
END_VAR
VAR_IN_OUT
	CheckPos												:	KIN_POSITIONS_MCS_DUT;
	Window													:	KIN_POSITIONS_MCS_DUT;
END_VAR                 									
VAR CONSTANT            									
END_VAR
isInPosExt													:= (CAM(CheckPos.X, MCS.X ,Window.X) OR NOT Config.0)
																AND (CAM(CheckPos.Y, MCS.Y ,Window.Y) OR NOT Config.1)
																AND (CAM(CheckPos.Z, MCS.Z ,Window.Z) OR NOT Config.2)
																AND (CAM(CheckPos.A, MCS.A ,Window.A) OR NOT Config.3)
																AND (CAM(CheckPos.B, MCS.B ,Window.B) OR NOT Config.4)
																AND (CAM(CheckPos.C, MCS.C ,Window.C) OR NOT Config.5)
																AND (CAM(CheckPos.Q1, MCS.Q1 ,Window.Q1) OR NOT Config.6)
																AND (CAM(CheckPos.Q2, MCS.Q2 ,Window.Q2) OR NOT Config.7);
END_METHOD

METHOD PUBLIC isInPosXYZ : BOOL //Return value = TRUE if axes are within window of checkPos values
VAR_IN_OUT
	CheckPos												:	KIN_POSITIONS_MCS_DUT;
	Window													:	KIN_POSITIONS_MCS_DUT;
END_VAR                 									
VAR CONSTANT            									
END_VAR
IsInPosXYZ												 	:= CAM(CheckPos.X, MCS.X ,Window.X)
																AND CAM(CheckPos.Y, MCS.Y ,Window.Y)
																AND CAM(CheckPos.Z, MCS.Z ,Window.Z);
END_METHOD

METHOD PUBLIC reset : BOOL //Delete data and reset valid , TRUE if execution finished
VAR_INPUT
END_VAR
Delete(); 
Valid														:= FALSE;
reset														:= TRUE;
END_METHOD

END_FUNCTION_BLOCK

// POUs/Motion/TF511x-KIN/03_DUTs/Trafo/KIN_CALCTRAFO_AXPOS_PARAM
FUNCTION_BLOCK KIN_CALCTRAFO_AXPOS_PARAM
VAR_INPUT
	In														: 	ARRAY[1..8] OF LREAL;
	Out														: 	ARRAY[1..8] OF LREAL;
	MetaInfoIn												:	U_KinMetaInfo;
	MetaInfoOut												:	U_KinMetaInfo;
END_VAR
VAR_OUTPUT
END_VAR
VAR
END_VAR

METHOD delete : BOOL
VAR_INPUT
END_VAR
MEMSET(ADR(In),0,SIZEOF(In));
MEMSET(ADR(Out),0,SIZEOF(Out));
delete	:= TRUE;
END_METHOD

END_FUNCTION_BLOCK

// POUs/Motion/TF511x-KIN/03_DUTs/Trafo/KIN_STATE_OBSERVER_OID_PARAM
{attribute 'hide'}
FUNCTION_BLOCK KIN_STATE_OBSERVER_OID_PARAM
VAR_INPUT
	oid														:	UDINT := 0; (* Scara State Observer OID *)
	TooltrafoOID											:	UDINT := 0; (* ToolTrafoOID *)
	NextTrafoOID											:	UDINT := 0; (*StaticTrafoOID *)

END_VAR
VAR_OUTPUT

END_VAR
VAR
END_VAR

;

METHOD delete : BOOL
VAR_INPUT
END_VAR
	oid														:= 0;
	TooltrafoOID											:= 0;
	NextTrafoOID											:= 0;
delete	:= TRUE;
END_METHOD

END_FUNCTION_BLOCK

// POUs/Motion/TF511x-KIN/03_DUTs/Trafo/KIN_STATICTRAFO_PARAM
{attribute 'hide'}
FUNCTION_BLOCK KIN_STATICTRAFO_PARAM
VAR_INPUT
	oid														:	UDINT := 0;
	TranslationX											:	LREAL := 0.0;
	TranslationY											:	LREAL := 0.0;
	TranslationZ											:	LREAL := 0.0;
                            								
	Rotation												: LREAL := 0.0;
	RotationAxis											: INT := 2;

END_VAR
VAR_OUTPUT

END_VAR
VAR
END_VAR

;

METHOD delete : BOOL
VAR_INPUT
END_VAR
	oid														:= 0;
	TranslationX											:= 0.0;
	TranslationY											:= 0.0;
	TranslationZ											:= 0.0;
                            								
	Rotation												:= 0.0;
	RotationAxis											:= 2;
delete	:= TRUE;
END_METHOD

END_FUNCTION_BLOCK

// POUs/Motion/TF511x-KIN/03_DUTs/Trafo/KIN_TOOLTRAFO_PARAM
{attribute 'hide'}
FUNCTION_BLOCK KIN_TOOLTRAFO_PARAM
VAR_INPUT
	oid														:	UDINT := 0;
	dx														: 	LREAL := 0.0;  (* Default Tooldata at WOS *)
	dy														: 	LREAL := 0.0;  (* Default Tooldata at WOS *)
	dz														:	LREAL := 0.0;  (* Default Tooldata at WOS *)

END_VAR
VAR_OUTPUT

END_VAR
VAR
END_VAR

;

METHOD delete : BOOL
VAR_INPUT
END_VAR
	oid														:= 0;
	dx														:= 0.0;  (* Default Tooldata at WOS *)
	dy														:= 0.0;  (* Default Tooldata at WOS *)
	dz														:= 0.0;  (* Default Tooldata at WOS *)
delete	:= TRUE;
END_METHOD

END_FUNCTION_BLOCK

// POUs/Motion/TF511x-KIN/KinChannel
FUNCTION_BLOCK KinChannel EXTENDS KIN_REF
VAR_INPUT
	Admin													:	KinAdmin;
END_VAR
VAR_OUTPUT
END_VAR
VAR
END_VAR

(* Kinematic Ctrl 										*)
(********************************************************)

(* work IO ********************************************************************)
(*	IO(); *)
	
(****************************************************************************)
(* Kinematic group control													*)
(****************************************************************************)
	Admin(
		ResetTrig			:= ,
		Enable			:= ,
		Override		:= ,
		ItpChannelId	:= ,
		AxesList		:= ,
		rKINRef			:= THIS^,
		Busy			=> ,
		Done			=> ,
		Error			=> ,
		ErrorId			=> );
(****************************************************************************)

END_FUNCTION_BLOCK

// POUs/Motion/VALUE_3D
{attribute 'no_check'}
FUNCTION_BLOCK VALUE_3D
VAR_INPUT                                                            
	Valid													:	BOOL ;
	X														:	LREAL;
	Y														:	LREAL;
	Z														:	LREAL;
END_VAR
VAR_OUTPUT
END_VAR
VAR
END_VAR

;

METHOD PUBLIC copy : BOOL //Return value = TRUE if execution finished
VAR_IN_OUT
	Source													:	VALUE_3D;
END_VAR
	Valid													:= Source.Valid;
	X														:= Source.X;
	Y														:= Source.Y;
	Z														:= Source.Z;
	copy													:= TRUE;
END_METHOD

METHOD PUBLIC delete : BOOL //Return value = TRUE if execution finished - Valid bit will not change
VAR_INPUT
END_VAR
	X					 									:= 0.0;	
	Y					 									:= 0.0;	
	Z					 									:= 0.0;	
	delete													:= TRUE;
END_METHOD

METHOD PUBLIC InPos : BOOL //Return value = TRUE axes is within window of checkPos values
VAR_IN_OUT
	CheckPos												:	VALUE_3D;
	Window													:	VALUE_3D;
END_VAR
InPos														:= CAM(CheckPos.X, X ,Window.X)
																AND CAM(CheckPos.Y, Y ,Window.Y)
																AND CAM(CheckPos.Z, Z ,Window.Z);
END_METHOD

METHOD PUBLIC InPosByAxisNo : BOOL //Return value = TRUE selected axis is within window of checkPos values
VAR_INPUT
	No					:	INT;
END_VAR
VAR_IN_OUT
	CheckPos			:	VALUE_3D;
	Window				:	VALUE_3D;
END_VAR
InPosByAxisNo													:= (CAM(CheckPos.X, X ,Window.X) OR No <> 1)
																AND (CAM(CheckPos.Y, Y ,Window.Y) OR No <> 2)
																AND (CAM(CheckPos.Z, Z ,Window.Z) OR No <> 3);
END_METHOD

METHOD PUBLIC InPosXY : BOOL //Return value = TRUE if axes are within window of checkPos values
VAR_IN_OUT
	CheckPos			:	VALUE_3D;
	Window				:	VALUE_3D;
END_VAR
InPosXY 													:= CAM(CheckPos.X, X ,Window.X)
																AND CAM(CheckPos.Y, Y ,Window.Y);
END_METHOD

METHOD PUBLIC InPosXZ : BOOL //Return value = TRUE if axes are within window of checkPos values
VAR_IN_OUT
	CheckPos			:	VALUE_3D;
	Window				:	VALUE_3D;
	
END_VAR
InPosXZ														:= CAM(CheckPos.X, X ,Window.X)
																AND CAM(CheckPos.Z, Z ,Window.Z);
END_METHOD

METHOD PUBLIC InPosYZ : BOOL //Return value = TRUE if axes are within window of checkPos values
VAR_IN_OUT
	CheckPos			:	VALUE_3D;
	Window				:	VALUE_3D;
	
END_VAR
InPosYZ													:= CAM(CheckPos.Y, Y ,Window.Y)
																AND CAM(CheckPos.Z, Z ,Window.Z);
END_METHOD

METHOD PUBLIC reset : BOOL //Delete data and reset valid , TRUE if execution finished
VAR_INPUT
END_VAR
Delete();
Valid														:= FALSE;
reset														:= TRUE;
END_METHOD

END_FUNCTION_BLOCK

// POUs/Motion/VALUE_6D
{attribute 'no_check'}
FUNCTION_BLOCK VALUE_6D 
VAR_INPUT
	Valid													:	BOOL ;
	X														:	LREAL;
	Y														:	LREAL;
	Z														:	LREAL;
	A														:		LREAL; //Rx
	B														:		LREAL; //Ry
	C														:		LREAL; //Rz	
END_VAR
VAR_OUTPUT
END_VAR
VAR
END_VAR

;

METHOD PUBLIC copy : BOOL //Return value = TRUE if execution finished
VAR_IN_OUT
	Source													:	VALUE_6D;
END_VAR
	Valid													:= Source.Valid;
	X														:= Source.X;
	Y														:= Source.Y;
	Z														:= Source.Z;
	A														:= Source.A;
	B														:= Source.B;
	C														:= Source.C;
	copy													:= TRUE;
END_METHOD

METHOD PUBLIC delete : BOOL //Return value = TRUE if execution finished - Valid bit will not change
VAR_INPUT
END_VAR
	X					 									:= 0.0;	
	Y					 									:= 0.0;	
	Z					 									:= 0.0;	
	A						 								:= 0.0;	
	B						 								:= 0.0;	
	C						 								:= 0.0;	
	delete													:= TRUE;
END_METHOD

METHOD PUBLIC inPos : BOOL //Return value = TRUE if axes are within window of checkPos values
VAR_IN_OUT
	CheckPos												:	VALUE_6D;
	Window													:	VALUE_6D;
END_VAR             										
VAR CONSTANT        										
END_VAR
InPos 														:= CAM(CheckPos.X, X, Window.X)
																AND CAM(CheckPos.Y, Y ,Window.Y)
																AND CAM(CheckPos.Z, Z,Window.Z)
																AND CAM(CheckPos.A, A, Window.A)
																AND CAM(CheckPos.B, B ,Window.B)
																AND CAM(CheckPos.C, C,Window.C);
END_METHOD

METHOD PUBLIC InPosABC : BOOL //Return value = TRUE if axes are within window of checkPos values
VAR_IN_OUT
	CheckPos												:	VALUE_6D;
	Window													:	VALUE_6D;
END_VAR                 									
VAR CONSTANT            									
END_VAR
InPosABC												 	:= CAM(CheckPos.A, A ,Window.A)
																AND CAM(CheckPos.B, B ,Window.B)
																AND CAM(CheckPos.C, C ,Window.C);
END_METHOD

METHOD PUBLIC InPosAC : BOOL //Return value = TRUE if axes are within window of checkPos values
VAR_IN_OUT
	CheckPos												:	VALUE_6D;
	Window													:	VALUE_6D;
END_VAR                 									
VAR CONSTANT            									
END_VAR
InPosAC													 	:= CAM(CheckPos.A, A ,Window.A)
																AND CAM(CheckPos.C, C ,Window.C);
END_METHOD

METHOD PUBLIC inPosByAxisNo : BOOL //Return value = TRUE selected axis is within window of checkPos values
VAR_INPUT
	No					:	INT;
END_VAR
VAR_IN_OUT
	CheckPos			:	VALUE_6D;
	Window				:	VALUE_6D;
END_VAR
inPosByAxisNo													:= (CAM(CheckPos.X, X ,Window.X) OR No <> 1)
																AND (CAM(CheckPos.Y, Y ,Window.Y) OR No <> 2)
																AND (CAM(CheckPos.Z, Z ,Window.Z) OR No <> 3)
																AND (CAM(CheckPos.A, A ,Window.A) OR No <> 4)
																AND (CAM(CheckPos.B, B ,Window.B) OR No <> 5)
																AND (CAM(CheckPos.C, C ,Window.C) OR No <> 6);
END_METHOD

